C05469=1228.924,245.140,-60.585,-176.917,6.303,148.228
C05470=1228.928,244.891,-60.559,-176.919,6.301,148.228
C05471=1228.932,244.643,-60.532,-176.921,6.299,148.228
C05472=1228.937,244.394,-60.506,-176.924,6.297,148.229
C05473=1228.941,244.145,-60.480,-176.927,6.295,148.229
C05474=1228.945,243.897,-60.454,-176.929,6.293,148.229
C05475=1228.950,243.648,-60.428,-176.932,6.291,148.230
C05476=1228.955,243.399,-60.402,-176.934,6.289,148.230
C05477=1228.959,243.151,-60.376,-176.937,6.287,148.230
C05478=1228.963,242.902,-60.349,-176.939,6.285,148.230
C05479=1228.968,242.653,-60.323,-176.941,6.284,148.231
C05480=1228.972,242.405,-60.297,-176.944,6.282,148.231
C05481=1228.976,242.157,-60.272,-176.946,6.280,148.231
C05482=1228.981,241.908,-60.245,-176.949,6.278,148.231
C05483=1228.986,241.659,-60.220,-176.951,6.276,148.232
C05484=1228.990,241.411,-60.193,-176.954,6.275,148.232
C05485=1228.995,241.162,-60.167,-176.956,6.273,148.232
C05486=1228.999,240.914,-60.141,-176.959,6.271,148.233
C05487=1229.004,240.665,-60.116,-176.961,6.269,148.233
C05488=1229.008,240.416,-60.090,-176.964,6.267,148.233
C05489=1229.012,240.168,-60.063,-176.966,6.265,148.233
C05490=1229.017,239.920,-60.037,-176.969,6.263,148.234
C05491=1229.022,239.671,-60.012,-176.972,6.261,148.234
C05492=1229.026,239.422,-59.986,-176.974,6.259,148.234
C05493=1229.030,239.173,-59.960,-176.977,6.257,148.235
C05494=1229.036,238.925,-59.934,-176.979,6.255,148.235
C05495=1229.040,238.676,-59.908,-176.982,6.253,148.235
C05496=1229.044,238.428,-59.882,-176.984,6.251,148.235
C05497=1229.048,238.179,-59.856,-176.987,6.250,148.236
C05498=1229.053,237.908,-59.828,-176.990,6.248,148.236
C05499=1229.058,237.636,-59.800,-176.992,6.246,148.236
C05500=1229.063,237.365,-59.772,-176.995,6.244,148.237
C05501=1229.068,237.093,-59.744,-176.997,6.242,148.237
C05502=1229.073,236.844,-59.718,-177.000,6.240,148.237
C05503=1229.077,236.596,-59.692,-177.003,6.238,148.238
C05504=1229.082,236.347,-59.667,-177.005,6.236,148.238
C05505=1229.086,236.099,-59.641,-177.008,6.235,148.238
C05506=1229.090,235.850,-59.615,-177.010,6.232,148.238
C05507=1229.095,235.602,-59.590,-177.013,6.230,148.239
C05508=1229.099,235.353,-59.564,-177.015,6.229,148.239
C05509=1229.103,235.104,-59.538,-177.018,6.227,148.239
C05510=1229.108,234.856,-59.513,-177.020,6.225,148.240
C05511=1229.113,234.607,-59.486,-177.023,6.223,148.240
C05512=1229.117,234.358,-59.461,-177.026,6.221,148.240
C05513=1229.122,234.110,-59.435,-177.028,6.219,148.241
C05514=1229.126,233.861,-59.410,-177.031,6.217,148.241
C05515=1229.131,233.612,-59.384,-177.032,6.216,148.241
C05516=1229.136,233.364,-59.359,-177.035,6.214,148.241
C05517=1229.140,233.115,-59.333,-177.038,6.212,148.242
C05518=1229.144,232.866,-59.308,-177.040,6.210,148.242
C05519=1229.149,232.618,-59.282,-177.043,6.208,148.242
C05520=1229.153,232.369,-59.256,-177.046,6.207,148.243
C05521=1229.157,232.120,-59.231,-177.048,6.205,148.243
C05522=1229.163,231.872,-59.206,-177.051,6.203,148.243
C05523=1229.167,231.623,-59.180,-177.053,6.201,148.244
C05524=1229.172,231.375,-59.155,-177.056,6.199,148.244
C05525=1229.176,231.126,-59.129,-177.059,6.197,148.244
C05526=1229.180,230.877,-59.103,-177.060,6.196,148.244
C05527=1229.185,230.628,-59.079,-177.063,6.194,148.245
C05528=1229.189,230.379,-59.053,-177.066,6.192,148.245
C05529=1229.194,230.131,-59.028,-177.068,6.190,148.245
C05530=1229.199,229.882,-59.003,-177.071,6.188,148.246
C05531=1229.202,229.633,-58.977,-177.073,6.186,148.246
C05532=1229.207,229.385,-58.952,-177.076,6.185,148.246
C05533=1229.211,229.137,-58.926,-177.079,6.183,148.247
C05534=1229.216,228.888,-58.902,-177.081,6.181,148.247
C05535=1229.221,228.639,-58.876,-177.084,6.179,148.247
C05536=1229.225,228.390,-58.850,-177.086,6.178,148.248
C05537=1229.230,228.141,-58.825,-177.089,6.176,148.248
C05538=1229.234,227.893,-58.800,-177.091,6.174,148.248
C05539=1229.239,227.645,-58.774,-177.094,6.172,148.249
C05540=1229.244,227.395,-58.749,-177.096,6.170,148.249
C05541=1229.248,227.147,-58.724,-177.099,6.168,148.249
C05542=1229.252,226.898,-58.699,-177.101,6.166,148.249
C05543=1229.257,226.650,-58.674,-177.104,6.165,148.250
C05544=1229.261,226.401,-58.648,-177.106,6.163,148.250
C05545=1229.266,226.152,-58.624,-177.108,6.162,148.250
C05546=1229.271,225.903,-58.598,-177.111,6.160,148.251
C05547=1229.274,225.654,-58.573,-177.114,6.158,148.251
C05548=1229.279,225.406,-58.548,-177.116,6.156,148.251
C05549=1229.284,225.157,-58.523,-177.119,6.154,148.252
C05550=1229.289,224.909,-58.498,-177.122,6.152,148.252
C05551=1229.293,224.659,-58.473,-177.124,6.150,148.252
C05552=1229.297,224.412,-58.448,-177.127,6.149,148.253
C05553=1229.302,224.162,-58.423,-177.129,6.147,148.253
C05554=1229.307,223.914,-58.397,-177.132,6.146,148.253
C05555=1229.311,223.665,-58.372,-177.134,6.144,148.254
C05556=1229.315,223.417,-58.348,-177.137,6.142,148.254
C05557=1229.320,223.168,-58.323,-177.139,6.140,148.254
C05558=1229.325,222.919,-58.297,-177.142,6.138,148.255
C05559=1229.330,222.671,-58.272,-177.145,6.136,148.255
C05560=1229.333,222.421,-58.248,-177.147,6.134,148.255
C05561=1229.338,222.173,-58.223,-177.149,6.133,148.256
C05562=1229.343,221.924,-58.198,-177.152,6.132,148.256
C05563=1229.348,221.676,-58.172,-177.155,6.130,148.256
C05564=1229.351,221.427,-58.148,-177.157,6.128,148.257
C05565=1229.357,221.178,-58.123,-177.160,6.126,148.257
C05566=1229.361,220.929,-58.097,-177.162,6.124,148.257
C05567=1229.365,220.681,-58.073,-177.165,6.122,148.258
C05568=1229.370,220.432,-58.049,-177.168,6.120,148.258
C05569=1229.375,220.183,-58.023,-177.170,6.119,148.258
C05570=1229.379,219.935,-57.999,-177.172,6.117,148.259
C05571=1229.384,219.685,-57.974,-177.175,6.116,148.259
C05572=1229.388,219.437,-57.950,-177.178,6.114,148.259
C05573=1229.392,219.188,-57.924,-177.180,6.112,148.260
C05574=1229.397,218.939,-57.899,-177.183,6.110,148.260
C05575=1229.402,218.691,-57.875,-177.186,6.108,148.260
C05576=1229.406,218.442,-57.850,-177.188,6.107,148.261
C05577=1229.411,218.193,-57.825,-177.190,6.105,148.261
C05578=1229.415,217.944,-57.800,-177.193,6.103,148.261
C05579=1229.420,217.696,-57.776,-177.196,6.101,148.262
C05580=1229.424,217.447,-57.752,-177.198,6.100,148.262
C05581=1229.429,217.198,-57.727,-177.201,6.098,148.262
C05582=1229.433,216.950,-57.702,-177.203,6.096,148.263
C05583=1229.438,216.701,-57.677,-177.205,6.095,148.263
C05584=1229.443,216.452,-57.652,-177.208,6.093,148.263
C05585=1229.447,216.203,-57.628,-177.211,6.091,148.264
C05586=1229.452,215.955,-57.603,-177.213,6.089,148.264
C05587=1229.456,215.706,-57.579,-177.216,6.087,148.264
C05588=1229.461,215.457,-57.554,-177.219,6.086,148.265
C05589=1229.465,215.209,-57.529,-177.221,6.085,148.265
C05590=1229.470,214.960,-57.504,-177.223,6.083,148.265
C05591=1229.474,214.711,-57.480,-177.226,6.081,148.266
C05592=1229.479,214.463,-57.456,-177.229,6.079,148.266
C05593=1229.483,214.213,-57.431,-177.232,6.077,148.266
C05594=1229.488,213.965,-57.407,-177.234,6.076,148.267
C05595=1229.493,213.716,-57.382,-177.236,6.074,148.267
C05596=1229.497,213.467,-57.357,-177.239,6.073,148.267
C05597=1229.501,213.218,-57.333,-177.242,6.071,148.268
C05598=1229.507,212.970,-57.309,-177.244,6.069,148.268
C05599=1229.510,212.721,-57.284,-177.247,6.067,148.268
C05600=1229.515,212.472,-57.260,-177.250,6.065,148.269
C05601=1229.520,212.223,-57.235,-177.252,6.064,148.269
C05602=1229.525,211.953,-57.209,-177.254,6.062,148.270
C05603=1229.530,211.682,-57.182,-177.257,6.061,148.270
C05604=1229.534,211.412,-57.156,-177.261,6.058,148.270
C05605=1229.539,211.142,-57.130,-177.263,6.056,148.271
C05606=1229.545,210.893,-57.105,-177.265,6.055,148.271
C05607=1229.548,210.644,-57.080,-177.268,6.053,148.271
C05608=1229.553,210.396,-57.056,-177.270,6.051,148.272
C05609=1229.558,210.147,-57.032,-177.273,6.050,148.272
C05610=1229.563,209.898,-57.008,-177.276,6.048,148.272
C05611=1229.566,209.649,-56.984,-177.278,6.047,148.273
C05612=1229.572,209.400,-56.959,-177.281,6.045,148.273
C05613=1229.576,209.152,-56.935,-177.284,6.043,148.274
C05614=1229.580,208.903,-56.911,-177.286,6.041,148.274
C05615=1229.585,208.654,-56.886,-177.289,6.040,148.274
C05616=1229.590,208.405,-56.863,-177.291,6.039,148.275
C05617=1229.594,208.156,-56.839,-177.294,6.037,148.275
C05618=1229.599,207.908,-56.814,-177.296,6.035,148.275
C05619=1229.603,207.659,-56.790,-177.299,6.033,148.276
C05620=1229.608,207.411,-56.766,-177.301,6.031,148.276
C05621=1229.613,207.161,-56.742,-177.304,6.030,148.276
C05622=1229.617,206.912,-56.717,-177.306,6.028,148.277
C05623=1229.621,206.664,-56.693,-177.309,6.027,148.277
C05624=1229.626,206.415,-56.670,-177.312,6.025,148.278
C05625=1229.631,206.166,-56.645,-177.314,6.024,148.278
C05626=1229.635,205.917,-56.621,-177.317,6.022,148.278
C05627=1229.640,205.669,-56.597,-177.319,6.020,148.279
C05628=1229.644,205.420,-56.573,-177.322,6.018,148.279
C05629=1229.649,205.171,-56.549,-177.325,6.016,148.279
C05630=1229.654,204.922,-56.525,-177.327,6.015,148.280
C05631=1229.658,204.673,-56.501,-177.329,6.014,148.280
C05632=1229.662,204.424,-56.477,-177.332,6.012,148.280
C05633=1229.667,204.176,-56.452,-177.335,6.010,148.281
C05634=1229.672,203.926,-56.429,-177.337,6.009,148.281
C05635=1229.676,203.678,-56.405,-177.340,6.007,148.282
C05636=1229.681,203.429,-56.381,-177.342,6.005,148.282
C05637=1229.686,203.181,-56.357,-177.345,6.004,148.282
C05638=1229.690,202.932,-56.333,-177.347,6.003,148.283
C05639=1229.695,202.683,-56.309,-177.350,6.001,148.283
C05640=1229.699,202.434,-56.285,-177.352,5.999,148.283
C05641=1229.704,202.185,-56.262,-177.355,5.997,148.284
C05642=1229.708,201.936,-56.237,-177.358,5.996,148.284
C05643=1229.713,201.687,-56.214,-177.360,5.994,148.285
C05644=1229.717,201.439,-56.190,-177.363,5.993,148.285
C05645=1229.722,201.190,-56.167,-177.365,5.991,148.285
C05646=1229.727,200.941,-56.142,-177.368,5.990,148.286
C05647=1229.732,200.692,-56.119,-177.370,5.988,148.286
C05648=1229.736,200.444,-56.095,-177.373,5.986,148.286
C05649=1229.741,200.195,-56.071,-177.376,5.984,148.287
C05650=1229.745,199.946,-56.047,-177.378,5.983,148.287
C05651=1229.749,199.696,-56.023,-177.381,5.982,148.288
C05652=1229.754,199.448,-55.999,-177.383,5.980,148.288
C05653=1229.759,199.199,-55.976,-177.386,5.978,148.288
C05654=1229.763,198.950,-55.953,-177.388,5.977,148.289
C05655=1229.768,198.702,-55.929,-177.391,5.975,148.289
C05656=1229.772,198.453,-55.905,-177.394,5.973,148.290
C05657=1229.777,198.204,-55.881,-177.396,5.972,148.290
C05658=1229.781,197.955,-55.858,-177.398,5.971,148.290
C05659=1229.786,197.706,-55.834,-177.401,5.969,148.291
C05660=1229.791,197.458,-55.810,-177.404,5.967,148.291
C05661=1229.795,197.209,-55.787,-177.406,5.966,148.291
C05662=1229.800,196.960,-55.764,-177.408,5.964,148.292
C05663=1229.804,196.711,-55.740,-177.412,5.962,148.292
C05664=1229.809,196.462,-55.716,-177.414,5.961,148.293
C05665=1229.814,196.213,-55.693,-177.416,5.960,148.293
C05666=1229.818,195.964,-55.669,-177.419,5.958,148.293
C05667=1229.823,195.716,-55.645,-177.422,5.956,148.294
C05668=1229.828,195.467,-55.622,-177.424,5.955,148.294
C05669=1229.832,195.218,-55.599,-177.427,5.953,148.295
C05670=1229.837,194.969,-55.575,-177.429,5.951,148.295
C05671=1229.841,194.720,-55.551,-177.432,5.950,148.295
C05672=1229.846,194.471,-55.528,-177.434,5.949,148.296
C05673=1229.851,194.222,-55.505,-177.437,5.947,148.296
C05674=1229.855,193.973,-55.481,-177.439,5.945,148.296
C05675=1229.860,193.725,-55.457,-177.442,5.944,148.297
C05676=1229.865,193.476,-55.434,-177.445,5.942,148.297
C05677=1229.869,193.227,-55.410,-177.447,5.941,148.298
C05678=1229.873,192.978,-55.388,-177.449,5.940,148.298
C05679=1229.878,192.729,-55.364,-177.452,5.938,148.298
C05680=1229.883,192.480,-55.341,-177.455,5.936,148.299
C05681=1229.888,192.232,-55.317,-177.457,5.935,148.299
C05682=1229.892,191.983,-55.294,-177.460,5.933,148.300
C05683=1229.897,191.734,-55.270,-177.463,5.931,148.300
C05684=1229.902,191.485,-55.247,-177.465,5.930,148.300
C05685=1229.906,191.236,-55.224,-177.467,5.929,148.301
C05686=1229.910,190.987,-55.201,-177.470,5.927,148.301
C05687=1229.915,190.738,-55.178,-177.473,5.925,148.302
C05688=1229.920,190.489,-55.154,-177.475,5.924,148.302
C05689=1229.924,190.240,-55.131,-177.478,5.922,148.302
C05690=1229.929,189.991,-55.108,-177.480,5.920,148.303
C05691=1229.933,189.742,-55.085,-177.483,5.920,148.303
C05692=1229.938,189.494,-55.062,-177.486,5.918,148.304
C05693=1229.943,189.245,-55.038,-177.488,5.916,148.304
C05694=1229.948,188.996,-55.015,-177.490,5.915,148.304
C05695=1229.953,188.747,-54.992,-177.493,5.913,148.305
C05696=1229.956,188.498,-54.969,-177.496,5.912,148.305
C05697=1229.961,188.249,-54.946,-177.498,5.911,148.306
C05698=1229.966,188.000,-54.922,-177.501,5.909,148.306
C05699=1229.971,187.751,-54.899,-177.503,5.907,148.306
C05700=1229.975,187.503,-54.876,-177.506,5.906,148.307
C05701=1229.980,187.254,-54.853,-177.509,5.904,148.307
C05702=1229.985,187.005,-54.830,-177.511,5.903,148.308
C05703=1229.989,186.756,-54.806,-177.513,5.902,148.308
C05704=1229.993,186.507,-54.784,-177.516,5.900,148.309
C05705=1229.998,186.258,-54.760,-177.519,5.899,148.309
C05706=1230.003,185.989,-54.735,-177.521,5.897,148.309
C05707=1230.008,185.719,-54.711,-177.524,5.895,148.310
C05708=1230.013,185.449,-54.686,-177.527,5.894,148.310
C05709=1230.018,185.180,-54.661,-177.530,5.892,148.311
C05710=1230.022,184.931,-54.638,-177.532,5.890,148.311
C05711=1230.028,184.682,-54.615,-177.535,5.890,148.312
C05712=1230.033,184.433,-54.592,-177.538,5.888,148.312
C05713=1230.037,184.184,-54.570,-177.540,5.886,148.312
C05714=1230.041,183.935,-54.546,-177.542,5.885,148.313
C05715=1230.046,183.686,-54.523,-177.545,5.883,148.313
C05716=1230.051,183.438,-54.500,-177.548,5.882,148.314
C05717=1230.056,183.188,-54.478,-177.550,5.880,148.314
C05718=1230.060,182.940,-54.455,-177.553,5.879,148.314
C05719=1230.064,182.691,-54.432,-177.555,5.878,148.315
C05720=1230.069,182.442,-54.408,-177.558,5.876,148.315
C05721=1230.074,182.193,-54.387,-177.561,5.874,148.316
C05722=1230.079,181.944,-54.363,-177.563,5.873,148.316
C05723=1230.083,181.695,-54.341,-177.566,5.872,148.317
C05724=1230.088,181.446,-54.318,-177.568,5.871,148.317
C05725=1230.092,181.198,-54.295,-177.571,5.869,148.317
C05726=1230.097,180.948,-54.272,-177.573,5.867,148.318
C05727=1230.102,180.699,-54.249,-177.576,5.866,148.318
C05728=1230.106,180.450,-54.227,-177.579,5.864,148.319
C05729=1230.111,180.202,-54.204,-177.581,5.863,148.319
C05730=1230.115,179.952,-54.182,-177.583,5.862,148.319
C05731=1230.120,179.703,-54.158,-177.586,5.860,148.320
C05732=1230.125,179.455,-54.136,-177.589,5.859,148.320
C05733=1230.130,179.206,-54.113,-177.591,5.857,148.321
C05734=1230.134,178.957,-54.091,-177.593,5.856,148.321
C05735=1230.139,178.707,-54.068,-177.596,5.855,148.322
C05736=1230.143,178.459,-54.045,-177.599,5.853,148.322
C05737=1230.148,178.210,-54.022,-177.601,5.852,148.323
C05738=1230.152,177.961,-54.000,-177.604,5.850,148.323
C05739=1230.157,177.713,-53.977,-177.606,5.849,148.323
C05740=1230.162,177.463,-53.955,-177.609,5.848,148.324
C05741=1230.166,177.214,-53.932,-177.612,5.846,148.324
C05742=1230.171,176.966,-53.910,-177.614,5.845,148.325
C05743=1230.175,176.717,-53.887,-177.617,5.843,148.325
C05744=1230.180,176.467,-53.865,-177.619,5.842,148.326
C05745=1230.185,176.219,-53.842,-177.622,5.840,148.326
C05746=1230.190,175.970,-53.820,-177.625,5.839,148.326
C05747=1230.194,175.721,-53.797,-177.627,5.838,148.327
C05748=1230.199,175.472,-53.774,-177.629,5.836,148.327
C05749=1230.204,175.223,-53.752,-177.632,5.835,148.328
C05750=1230.208,174.974,-53.730,-177.635,5.833,148.328
C05751=1230.213,174.725,-53.707,-177.637,5.832,148.329
C05752=1230.217,174.476,-53.685,-177.639,5.831,148.329
C05753=1230.222,174.227,-53.662,-177.643,5.829,148.330
C05754=1230.227,173.979,-53.640,-177.645,5.828,148.330
C05755=1230.231,173.729,-53.618,-177.647,5.826,148.330
C05756=1230.237,173.480,-53.595,-177.650,5.826,148.331
C05757=1230.241,173.231,-53.573,-177.653,5.824,148.331
C05758=1230.245,172.982,-53.550,-177.655,5.823,148.332
C05759=1230.250,172.733,-53.528,-177.657,5.821,148.332
C05760=1230.254,172.484,-53.505,-177.660,5.819,148.333
C05761=1230.259,172.236,-53.484,-177.663,5.818,148.333
C05762=1230.264,171.986,-53.461,-177.665,5.817,148.333
C05763=1230.268,171.737,-53.438,-177.668,5.816,148.334
C05764=1230.273,171.489,-53.417,-177.670,5.814,148.334
C05765=1230.278,171.239,-53.394,-177.673,5.813,148.335
C05766=1230.283,170.991,-53.372,-177.676,5.812,148.335
C05767=1230.287,170.742,-53.350,-177.678,5.811,148.336
C05768=1230.292,170.493,-53.328,-177.680,5.809,148.336
C05769=1230.297,170.244,-53.305,-177.684,5.807,148.337
C05770=1230.301,169.994,-53.283,-177.686,5.806,148.337
C05771=1230.306,169.746,-53.261,-177.688,5.804,148.337
C05772=1230.310,169.497,-53.239,-177.691,5.804,148.338
C05773=1230.316,169.248,-53.216,-177.694,5.802,148.338
C05774=1230.320,168.999,-53.194,-177.696,5.801,148.339
C05775=1230.325,168.750,-53.173,-177.698,5.799,148.339
C05776=1230.329,168.501,-53.150,-177.701,5.798,148.340
C05777=1230.334,168.252,-53.128,-177.704,5.797,148.340
C05778=1230.338,168.003,-53.106,-177.706,5.796,148.340
C05779=1230.343,167.754,-53.084,-177.709,5.794,148.341
C05780=1230.348,167.505,-53.062,-177.711,5.793,148.341
C05781=1230.352,167.256,-53.040,-177.714,5.791,148.342
C05782=1230.358,167.007,-53.018,-177.717,5.790,148.342
C05783=1230.362,166.758,-52.996,-177.719,5.789,148.343
C05784=1230.366,166.509,-52.973,-177.721,5.787,148.343
C05785=1230.371,166.261,-52.951,-177.724,5.786,148.344
C05786=1230.375,166.011,-52.929,-177.727,5.784,148.344
C05787=1230.380,165.763,-52.908,-177.729,5.784,148.345
C05788=1230.385,165.513,-52.885,-177.732,5.782,148.345
C05789=1230.390,165.264,-52.863,-177.734,5.781,148.345
C05790=1230.394,165.015,-52.841,-177.737,5.779,148.346
C05791=1230.399,164.766,-52.820,-177.739,5.778,148.346
C05792=1230.404,164.517,-52.798,-177.742,5.777,148.347
C05793=1230.408,164.268,-52.776,-177.744,5.776,148.347
C05794=1230.413,164.019,-52.754,-177.747,5.774,148.348
C05795=1230.418,163.770,-52.732,-177.749,5.773,148.348
C05796=1230.422,163.521,-52.710,-177.752,5.772,148.349
C05797=1230.427,163.272,-52.688,-177.754,5.771,148.349
C05798=1230.432,163.023,-52.666,-177.757,5.769,148.349
C05799=1230.437,162.774,-52.644,-177.760,5.768,148.350
C05800=1230.442,162.525,-52.622,-177.762,5.766,148.350
C05801=1230.446,162.276,-52.600,-177.764,5.765,148.351
C05802=1230.451,162.027,-52.579,-177.768,5.764,148.351
C05803=1230.455,161.778,-52.557,-177.770,5.763,148.352
C05804=1230.460,161.529,-52.536,-177.773,5.761,148.352
C05805=1230.465,161.280,-52.514,-177.775,5.760,148.353
C05806=1230.469,161.031,-52.492,-177.778,5.758,148.353
C05807=1230.474,160.782,-52.470,-177.780,5.758,148.354
C05808=1230.478,160.533,-52.448,-177.783,5.756,148.354
C05809=1230.483,160.284,-52.427,-177.785,5.755,148.355
C05810=1230.489,160.015,-52.403,-177.788,5.753,148.355
C05811=1230.493,159.746,-52.380,-177.791,5.752,148.356
C05812=1230.499,159.477,-52.356,-177.793,5.751,148.356
C05813=1230.503,159.208,-52.334,-177.797,5.749,148.357
C05814=1230.508,158.959,-52.312,-177.799,5.748,148.357
C05815=1230.513,158.710,-52.290,-177.801,5.747,148.358
C05816=1230.517,158.461,-52.268,-177.804,5.746,148.358
C05817=1230.522,158.211,-52.247,-177.807,5.744,148.358
C05818=1230.527,157.963,-52.225,-177.809,5.743,148.359
C05819=1230.531,157.714,-52.203,-177.812,5.742,148.359
C05820=1230.536,157.465,-52.181,-177.814,5.741,148.360
C05821=1230.541,157.216,-52.160,-177.817,5.739,148.360
C05822=1230.545,156.966,-52.138,-177.819,5.738,148.361
C05823=1230.550,156.718,-52.117,-177.822,5.737,148.361
C05824=1230.555,156.468,-52.096,-177.824,5.736,148.362
C05825=1230.560,156.219,-52.074,-177.826,5.735,148.362
C05826=1230.565,155.970,-52.052,-177.830,5.733,148.363
C05827=1230.569,155.721,-52.032,-177.832,5.732,148.363
C05828=1230.574,155.473,-52.010,-177.835,5.731,148.364
C05829=1230.578,155.223,-51.988,-177.837,5.730,148.364
C05830=1230.583,154.974,-51.967,-177.840,5.728,148.365
C05831=1230.588,154.726,-51.945,-177.842,5.727,148.365
C05832=1230.592,154.476,-51.923,-177.845,5.725,148.366
C05833=1230.598,154.227,-51.902,-177.848,5.725,148.366
C05834=1230.602,153.979,-51.881,-177.850,5.723,148.367
C05835=1230.606,153.729,-51.860,-177.852,5.722,148.367
C05836=1230.611,153.480,-51.838,-177.855,5.721,148.368
C05837=1230.616,153.231,-51.817,-177.858,5.719,148.368
C05838=1230.621,152.982,-51.796,-177.860,5.719,148.369
C05839=1230.626,152.733,-51.773,-177.863,5.717,148.369
C05840=1230.630,152.484,-51.753,-177.865,5.716,148.370
C05841=1230.635,152.235,-51.731,-177.868,5.714,148.370
C05842=1230.640,151.986,-51.710,-177.870,5.713,148.370
C05843=1230.644,151.737,-51.688,-177.873,5.712,148.371
C05844=1230.649,151.488,-51.668,-177.875,5.711,148.371
C05845=1230.654,151.239,-51.646,-177.878,5.710,148.372
C05846=1230.659,150.990,-51.625,-177.881,5.709,148.372
C05847=1230.663,150.740,-51.603,-177.883,5.708,148.373
C05848=1230.667,150.491,-51.583,-177.886,5.706,148.373
C05849=1230.672,150.243,-51.561,-177.888,5.705,148.374
C05850=1230.678,149.994,-51.540,-177.891,5.704,148.374
C05851=1230.682,149.744,-51.518,-177.893,5.703,148.375
C05852=1230.686,149.495,-51.498,-177.896,5.702,148.375
C05853=1230.691,149.246,-51.477,-177.899,5.700,148.376
C05854=1230.696,148.997,-51.455,-177.901,5.699,148.376
C05855=1230.701,148.748,-51.434,-177.904,5.698,148.377
C05856=1230.705,148.499,-51.413,-177.906,5.697,148.377
C05857=1230.710,148.250,-51.392,-177.908,5.696,148.378
C05858=1230.715,148.001,-51.371,-177.911,5.694,148.378
C05859=1230.719,147.752,-51.350,-177.914,5.693,148.379
C05860=1230.725,147.503,-51.329,-177.916,5.692,148.379
C05861=1230.730,147.254,-51.308,-177.919,5.691,148.380
C05862=1230.733,147.005,-51.286,-177.921,5.690,148.380
C05863=1230.739,146.755,-51.265,-177.924,5.689,148.381
C05864=1230.744,146.506,-51.245,-177.926,5.688,148.381
C05865=1230.748,146.258,-51.223,-177.930,5.686,148.382
C05866=1230.753,146.009,-51.202,-177.932,5.685,148.382
C05867=1230.757,145.760,-51.182,-177.934,5.684,148.383
C05868=1230.762,145.510,-51.160,-177.937,5.683,148.383
C05869=1230.767,145.261,-51.139,-177.939,5.682,148.384
C05870=1230.771,145.012,-51.119,-177.942,5.680,148.384
C05871=1230.776,144.763,-51.098,-177.944,5.679,148.385
C05872=1230.781,144.514,-51.077,-177.947,5.678,148.385
C05873=1230.786,144.265,-51.056,-177.950,5.677,148.386
C05874=1230.790,144.016,-51.035,-177.952,5.676,148.386
C05875=1230.795,143.766,-51.014,-177.955,5.674,148.387
C05876=1230.800,143.517,-50.993,-177.957,5.674,148.387
C05877=1230.804,143.269,-50.972,-177.959,5.673,148.388
C05878=1230.809,143.019,-50.951,-177.963,5.671,148.388
C05879=1230.814,142.771,-50.931,-177.965,5.670,148.389
C05880=1230.819,142.521,-50.910,-177.967,5.669,148.389
C05881=1230.823,142.272,-50.889,-177.970,5.668,148.390
C05882=1230.829,142.023,-50.868,-177.973,5.667,148.390
C05883=1230.833,141.775,-50.847,-177.975,5.665,148.391
C05884=1230.838,141.525,-50.826,-177.978,5.665,148.391
C05885=1230.842,141.276,-50.805,-177.980,5.664,148.392
C05886=1230.847,141.027,-50.785,-177.983,5.662,148.392
C05887=1230.851,140.778,-50.764,-177.985,5.661,148.393
C05888=1230.856,140.528,-50.743,-177.987,5.660,148.393
C05889=1230.861,140.279,-50.723,-177.991,5.659,148.394
C05890=1230.866,140.030,-50.702,-177.993,5.658,148.394
C05891=1230.870,139.781,-50.681,-177.996,5.656,148.395
C05892=1230.876,139.532,-50.660,-177.998,5.655,148.395
C05893=1230.880,139.283,-50.640,-178.000,5.655,148.396
C05894=1230.885,139.034,-50.619,-178.003,5.653,148.396
C05895=1230.890,138.785,-50.599,-178.006,5.652,148.397
C05896=1230.894,138.536,-50.578,-178.008,5.651,148.397
C05897=1230.899,138.287,-50.557,-178.011,5.650,148.398
C05898=1230.904,138.038,-50.537,-178.013,5.649,148.398
C05899=1230.909,137.788,-50.516,-178.016,5.648,148.399
C05900=1230.913,137.539,-50.496,-178.018,5.646,148.399
C05901=1230.919,137.290,-50.475,-178.021,5.646,148.400
C05902=1230.923,137.041,-50.454,-178.023,5.645,148.400
C05903=1230.927,136.792,-50.434,-178.026,5.643,148.401
C05904=1230.933,136.543,-50.413,-178.028,5.642,148.401
C05905=1230.937,136.294,-50.393,-178.031,5.641,148.402
C05906=1230.941,136.045,-50.372,-178.034,5.640,148.402
C05907=1230.947,135.796,-50.351,-178.036,5.639,148.403
C05908=1230.951,135.547,-50.331,-178.039,5.638,148.403
C05909=1230.956,135.298,-50.311,-178.042,5.637,148.404
C05910=1230.961,135.049,-50.290,-178.044,5.636,148.404
C05911=1230.965,134.799,-50.270,-178.046,5.635,148.405
C05912=1230.971,134.550,-50.249,-178.049,5.633,148.405
C05913=1230.975,134.301,-50.229,-178.052,5.632,148.406
C05914=1230.980,134.033,-50.206,-178.055,5.631,148.406
C05915=1230.985,133.763,-50.185,-178.057,5.630,148.407
C05916=1230.990,133.495,-50.162,-178.060,5.628,148.407
C05917=1230.996,133.226,-50.141,-178.063,5.628,148.408
C05918=1231.000,132.977,-50.120,-178.065,5.627,148.409
C05919=1231.005,132.728,-50.100,-178.068,5.625,148.409
C05920=1231.010,132.479,-50.079,-178.070,5.625,148.410
C05921=1231.014,132.230,-50.059,-178.073,5.624,148.410
C05922=1231.019,131.980,-50.039,-178.076,5.622,148.411
C05923=1231.023,131.731,-50.019,-178.078,5.621,148.411
C05924=1231.029,131.482,-49.998,-178.080,5.621,148.412
C05925=1231.033,131.233,-49.977,-178.083,5.619,148.412
C05926=1231.038,130.984,-49.958,-178.086,5.618,148.413
C05927=1231.043,130.735,-49.938,-178.088,5.617,148.413
C05928=1231.048,130.486,-49.917,-178.091,5.616,148.414
C05929=1231.053,130.236,-49.897,-178.094,5.615,148.414
C05930=1231.057,129.987,-49.877,-178.096,5.614,148.415
C05931=1231.062,129.739,-49.856,-178.099,5.613,148.415
C05932=1231.066,129.490,-49.836,-178.101,5.612,148.416
C05933=1231.071,129.240,-49.816,-178.104,5.611,148.417
C05934=1231.076,128.991,-49.795,-178.106,5.610,148.417
C05935=1231.081,128.742,-49.776,-178.109,5.609,148.418
C05936=1231.086,128.493,-49.756,-178.111,5.608,148.418
C05937=1231.090,128.244,-49.735,-178.114,5.607,148.419
C05938=1231.095,127.994,-49.716,-178.116,5.605,148.419
C05939=1231.100,127.745,-49.695,-178.119,5.605,148.420
C05940=1231.104,127.496,-49.674,-178.121,5.604,148.420
C05941=1231.109,127.247,-49.655,-178.124,5.603,148.421
C05942=1231.114,126.998,-49.634,-178.127,5.601,148.421
C05943=1231.119,126.749,-49.615,-178.129,5.601,148.422
C05944=1231.123,126.500,-49.595,-178.131,5.600,148.422
C05945=1231.128,126.250,-49.575,-178.134,5.598,148.423
C05946=1231.133,126.001,-49.554,-178.137,5.597,148.423
C05947=1231.138,125.751,-49.534,-178.139,5.597,148.424
C05948=1231.143,125.503,-49.514,-178.141,5.596,148.424
C05949=1231.148,125.254,-49.495,-178.145,5.594,148.425
C05950=1231.152,125.005,-49.474,-178.147,5.593,148.425
C05951=1231.157,124.755,-49.455,-178.149,5.593,148.426
C05952=1231.162,124.506,-49.434,-178.152,5.591,148.426
C05953=1231.166,124.257,-49.415,-178.155,5.590,148.427
C05954=1231.171,124.008,-49.395,-178.157,5.590,148.428
C05955=1231.176,123.759,-49.375,-178.159,5.589,148.428
C05956=1231.180,123.510,-49.354,-178.163,5.587,148.429
C05957=1231.185,123.260,-49.335,-178.165,5.586,148.429
C05958=1231.190,123.011,-49.314,-178.167,5.586,148.430
C05959=1231.195,122.762,-49.295,-178.170,5.585,148.430
C05960=1231.199,122.514,-49.275,-178.173,5.583,148.431
C05961=1231.204,122.264,-49.255,-178.175,5.583,148.431
C05962=1231.209,122.014,-49.235,-178.177,5.582,148.432
C05963=1231.214,121.766,-49.215,-178.180,5.581,148.432
C05964=1231.219,121.517,-49.196,-178.183,5.579,148.433
C05965=1231.223,121.267,-49.176,-178.185,5.579,148.434
C05966=1231.228,121.018,-49.156,-178.188,5.578,148.434
C05967=1231.233,120.769,-49.136,-178.190,5.577,148.435
C05968=1231.238,120.520,-49.117,-178.193,5.575,148.435
C05969=1231.242,120.271,-49.096,-178.195,5.574,148.436
C05970=1231.247,120.021,-49.077,-178.198,5.574,148.436
C05971=1231.252,119.772,-49.058,-178.200,5.573,148.437
C05972=1231.257,119.523,-49.037,-178.203,5.571,148.437
C05973=1231.262,119.274,-49.017,-178.206,5.571,148.438
C05974=1231.266,119.024,-48.998,-178.208,5.570,148.438
C05975=1231.271,118.776,-48.978,-178.210,5.569,148.439
C05976=1231.276,118.526,-48.958,-178.214,5.568,148.440
C05977=1231.281,118.277,-48.939,-178.216,5.567,148.440
C05978=1231.286,118.028,-48.919,-178.218,5.566,148.441
C05979=1231.291,117.779,-48.899,-178.220,5.565,148.441
C05980=1231.295,117.530,-48.880,-178.224,5.564,148.442
C05981=1231.300,117.281,-48.861,-178.226,5.563,148.442
C05982=1231.305,117.031,-48.841,-178.228,5.562,148.443
C05983=1231.310,116.782,-48.821,-178.231,5.561,148.443
C05984=1231.314,116.533,-48.801,-178.234,5.560,148.444
C05985=1231.319,116.284,-48.782,-178.236,5.559,148.444
C05986=1231.324,116.034,-48.762,-178.239,5.558,148.445
C05987=1231.329,115.785,-48.742,-178.241,5.557,148.445
C05988=1231.333,115.536,-48.724,-178.244,5.557,148.446
C05989=1231.338,115.287,-48.704,-178.247,5.555,148.447
C05990=1231.343,115.038,-48.684,-178.249,5.554,148.447
C05991=1231.348,114.789,-48.664,-178.251,5.554,148.448
C05992=1231.353,114.539,-48.645,-178.254,5.553,148.448
C05993=1231.358,114.290,-48.625,-178.257,5.551,148.449
C05994=1231.362,114.041,-48.606,-178.259,5.551,148.449
C05995=1231.367,113.792,-48.587,-178.261,5.550,148.450
C05996=1231.372,113.543,-48.567,-178.264,5.549,148.450
C05997=1231.377,113.293,-48.548,-178.267,5.548,148.451
C05998=1231.382,113.044,-48.528,-178.269,5.547,148.452
C05999=1231.386,112.795,-48.509,-178.272,5.546,148.452
C06000=1231.391,112.545,-48.490,-178.275,5.545,148.453
C06001=1231.396,112.297,-48.470,-178.277,5.544,148.453
C06002=1231.401,112.048,-48.450,-178.279,5.544,148.454
C06003=1231.405,111.798,-48.431,-178.283,5.542,148.454
C06004=1231.410,111.549,-48.412,-178.285,5.541,148.455
C06005=1231.415,111.300,-48.392,-178.287,5.541,148.456
C06006=1231.420,111.051,-48.373,-178.290,5.540,148.456
C06007=1231.424,110.802,-48.354,-178.292,5.539,148.457
C06008=1231.429,110.552,-48.335,-178.295,5.538,148.457
C06009=1231.435,110.303,-48.315,-178.297,5.537,148.458
C06010=1231.439,110.053,-48.296,-178.300,5.536,148.458
C06011=1231.444,109.805,-48.277,-178.302,5.536,148.459
C06012=1231.449,109.555,-48.257,-178.305,5.535,148.459
C06013=1231.454,109.306,-48.238,-178.308,5.533,148.460
C06014=1231.458,109.057,-48.219,-178.310,5.532,148.461
C06015=1231.463,108.807,-48.199,-178.313,5.532,148.461
C06016=1231.468,108.558,-48.180,-178.315,5.531,148.462
C06017=1231.472,108.309,-48.161,-178.318,5.530,148.462
C06018=1231.478,108.041,-48.140,-178.321,5.529,148.463
C06019=1231.483,107.772,-48.120,-178.323,5.528,148.463
C06020=1231.488,107.504,-48.099,-178.326,5.527,148.464
C06021=1231.493,107.235,-48.078,-178.329,5.526,148.465
C06022=1231.498,106.987,-48.059,-178.331,5.525,148.465
C06023=1231.503,106.737,-48.040,-178.334,5.525,148.466
C06024=1231.508,106.488,-48.021,-178.336,5.524,148.466
C06025=1231.512,106.239,-48.002,-178.339,5.523,148.467
C06026=1231.518,105.990,-47.983,-178.342,5.522,148.468
C06027=1231.522,105.740,-47.963,-178.344,5.521,148.468
C06028=1231.526,105.491,-47.944,-178.347,5.520,148.469
C06029=1231.532,105.241,-47.925,-178.349,5.519,148.469
C06030=1231.536,104.992,-47.906,-178.351,5.518,148.470
C06031=1231.541,104.743,-47.887,-178.354,5.518,148.470
C06032=1231.546,104.495,-47.868,-178.357,5.516,148.471
C06033=1231.551,104.244,-47.850,-178.359,5.515,148.471
C06034=1231.556,103.996,-47.830,-178.362,5.515,148.472
C06035=1231.560,103.746,-47.811,-178.365,5.514,148.473
C06036=1231.566,103.497,-47.792,-178.367,5.513,148.473
C06037=1231.570,103.248,-47.774,-178.369,5.512,148.474
C06038=1231.575,102.999,-47.754,-178.373,5.511,148.474
C06039=1231.579,102.749,-47.735,-178.375,5.510,148.475
C06040=1231.585,102.500,-47.717,-178.377,5.509,148.475
C06041=1231.589,102.251,-47.698,-178.380,5.509,148.476
C06042=1231.594,102.002,-47.678,-178.382,5.508,148.477
C06043=1231.599,101.752,-47.660,-178.385,5.507,148.477
C06044=1231.604,101.503,-47.641,-178.387,5.507,148.478
C06045=1231.609,101.255,-47.622,-178.390,5.505,148.478
C06046=1231.614,101.004,-47.603,-178.393,5.504,148.479
C06047=1231.618,100.756,-47.584,-178.395,5.504,148.480
C06048=1231.623,100.506,-47.565,-178.398,5.503,148.480
C06049=1231.628,100.257,-47.547,-178.400,5.502,148.481
C06050=1231.633,100.008,-47.527,-178.403,5.501,148.481
C06051=1231.638,99.758,-47.509,-178.405,5.501,148.482
C06052=1231.643,99.509,-47.490,-178.408,5.499,148.482
C06053=1231.647,99.260,-47.471,-178.410,5.498,148.483
C06054=1231.652,99.011,-47.453,-178.413,5.498,148.484
C06055=1231.657,98.761,-47.433,-178.416,5.497,148.484
C06056=1231.662,98.512,-47.415,-178.418,5.496,148.485
C06057=1231.667,98.263,-47.396,-178.420,5.496,148.485
C06058=1231.671,98.014,-47.377,-178.423,5.495,148.486
C06059=1231.677,97.765,-47.358,-178.425,5.494,148.486
C06060=1231.681,97.515,-47.340,-178.428,5.493,148.487
C06061=1231.685,97.266,-47.321,-178.431,5.492,148.488
C06062=1231.691,97.017,-47.302,-178.433,5.491,148.488
C06063=1231.695,96.768,-47.283,-178.436,5.490,148.489
C06064=1231.700,96.518,-47.265,-178.438,5.490,148.489
C06065=1231.705,96.269,-47.246,-178.441,5.489,148.490
C06066=1231.710,96.020,-47.228,-178.443,5.488,148.490
C06067=1231.715,95.770,-47.209,-178.446,5.488,148.491
C06068=1231.720,95.522,-47.191,-178.449,5.486,148.492
C06069=1231.724,95.272,-47.172,-178.451,5.486,148.492
C06070=1231.730,95.023,-47.153,-178.454,5.485,148.493
C06071=1231.734,94.774,-47.135,-178.456,5.484,148.493
C06072=1231.738,94.524,-47.116,-178.459,5.483,148.494
C06073=1231.744,94.275,-47.097,-178.461,5.482,148.495
C06074=1231.749,94.026,-47.079,-178.464,5.482,148.495
C06075=1231.753,93.776,-47.060,-178.466,5.481,148.496
C06076=1231.758,93.527,-47.042,-178.469,5.481,148.496
C06077=1231.764,93.278,-47.024,-178.472,5.479,148.497
C06078=1231.768,93.029,-47.005,-178.474,5.478,148.498
C06079=1231.773,92.779,-46.987,-178.477,5.478,148.498
C06080=1231.778,92.530,-46.968,-178.479,5.477,148.499
C06081=1231.782,92.281,-46.949,-178.482,5.476,148.499
C06082=1231.787,92.031,-46.931,-178.484,5.475,148.500
C06083=1231.792,91.782,-46.913,-178.487,5.475,148.501
C06084=1231.797,91.533,-46.893,-178.489,5.474,148.501
C06085=1231.802,91.284,-46.875,-178.492,5.473,148.502
C06086=1231.807,91.034,-46.857,-178.494,5.473,148.502
C06087=1231.811,90.785,-46.839,-178.497,5.471,148.503
C06088=1231.816,90.536,-46.820,-178.499,5.470,148.503
C06089=1231.821,90.286,-46.802,-178.502,5.470,148.504
C06090=1231.826,90.037,-46.784,-178.505,5.469,148.505
C06091=1231.831,89.788,-46.766,-178.507,5.468,148.505
C06092=1231.835,89.539,-46.747,-178.509,5.467,148.506
C06093=1231.841,89.289,-46.728,-178.512,5.467,148.506
C06094=1231.846,89.040,-46.710,-178.515,5.466,148.507
C06095=1231.850,88.791,-46.692,-178.517,5.466,148.508
C06096=1231.855,88.541,-46.674,-178.519,5.465,148.508
C06097=1231.859,88.293,-46.655,-178.522,5.464,148.509
C06098=1231.865,88.043,-46.637,-178.525,5.463,148.509
C06099=1231.870,87.794,-46.619,-178.528,5.462,148.510
C06100=1231.874,87.544,-46.600,-178.530,5.461,148.511
C06101=1231.879,87.295,-46.582,-178.533,5.460,148.511
C06102=1231.884,87.046,-46.564,-178.535,5.460,148.512
C06103=1231.889,86.797,-46.546,-178.538,5.459,148.512
C06104=1231.894,86.548,-46.528,-178.540,5.459,148.513
C06105=1231.899,86.298,-46.509,-178.543,5.458,148.514
C06106=1231.904,86.049,-46.491,-178.545,5.457,148.514
C06107=1231.908,85.799,-46.473,-178.548,5.457,148.515
C06108=1231.913,85.550,-46.455,-178.550,5.456,148.515
C06109=1231.918,85.301,-46.437,-178.553,5.455,148.516
C06110=1231.923,85.051,-46.418,-178.555,5.454,148.517
C06111=1231.927,84.802,-46.401,-178.558,5.454,148.517
C06112=1231.932,84.553,-46.383,-178.560,5.453,148.518
C06113=1231.937,84.304,-46.365,-178.563,5.452,148.518
C06114=1231.942,84.054,-46.347,-178.566,5.451,148.519
C06115=1231.947,83.805,-46.329,-178.568,5.450,148.520
C06116=1231.952,83.555,-46.310,-178.571,5.450,148.520
C06117=1231.957,83.306,-46.292,-178.574,5.449,148.521
C06118=1231.962,83.057,-46.274,-178.576,5.448,148.521
C06119=1231.967,82.808,-46.256,-178.578,5.447,148.522
C06120=1231.972,82.558,-46.238,-178.581,5.447,148.523
C06121=1231.977,82.309,-46.220,-178.584,5.446,148.523
C06122=1231.982,82.041,-46.200,-178.586,5.446,148.524
C06123=1231.987,81.773,-46.181,-178.589,5.445,148.525
C06124=1231.992,81.504,-46.162,-178.592,5.444,148.525
C06125=1231.997,81.236,-46.142,-178.595,5.443,148.526
C06126=1232.002,80.987,-46.124,-178.597,5.442,148.526
C06127=1232.006,80.737,-46.106,-178.599,5.441,148.527
C06128=1232.011,80.488,-46.088,-178.602,5.441,148.528
C06129=1232.016,80.238,-46.071,-178.605,5.440,148.528
C06130=1232.021,79.989,-46.053,-178.607,5.440,148.529
C06131=1232.026,79.740,-46.035,-178.610,5.439,148.529
C06132=1232.031,79.491,-46.017,-178.612,5.438,148.530
C06133=1232.036,79.241,-45.999,-178.615,5.437,148.531
C06134=1232.041,78.992,-45.981,-178.617,5.437,148.531
C06135=1232.046,78.743,-45.963,-178.620,5.436,148.532
C06136=1232.051,78.494,-45.945,-178.622,5.435,148.532
C06137=1232.055,78.243,-45.927,-178.625,5.435,148.533
C06138=1232.060,77.994,-45.909,-178.627,5.434,148.534
C06139=1232.065,77.745,-45.891,-178.630,5.434,148.534
C06140=1232.070,77.496,-45.873,-178.633,5.433,148.535
C06141=1232.075,77.247,-45.855,-178.635,5.432,148.536
C06142=1232.080,76.997,-45.838,-178.637,5.431,148.536
C06143=1232.084,76.748,-45.820,-178.640,5.431,148.537
C06144=1232.089,76.499,-45.803,-178.643,5.430,148.538
C06145=1232.094,76.250,-45.785,-178.645,5.430,148.538
C06146=1232.100,76.000,-45.767,-178.647,5.429,148.539
C06147=1232.104,75.751,-45.749,-178.650,5.428,148.539
C06148=1232.109,75.502,-45.731,-178.653,5.427,148.540
C06149=1232.114,75.252,-45.713,-178.655,5.427,148.541
C06150=1232.119,75.003,-45.697,-178.658,5.426,148.541
C06151=1232.124,74.754,-45.679,-178.660,5.425,148.542
C06152=1232.129,74.505,-45.661,-178.663,5.425,148.542
C06153=1232.133,74.255,-45.643,-178.665,5.424,148.543
C06154=1232.139,74.006,-45.625,-178.668,5.424,148.544
C06155=1232.144,73.756,-45.607,-178.671,5.423,148.544
C06156=1232.148,73.508,-45.590,-178.673,5.422,148.545
C06157=1232.153,73.258,-45.573,-178.675,5.421,148.545
C06158=1232.158,73.009,-45.555,-178.678,5.421,148.546
C06159=1232.163,72.759,-45.537,-178.681,5.420,148.547
C06160=1232.168,72.510,-45.520,-178.683,5.420,148.547
C06161=1232.172,72.261,-45.502,-178.686,5.419,148.548
C06162=1232.177,72.011,-45.485,-178.688,5.418,148.549
C06163=1232.182,71.762,-45.467,-178.691,5.418,148.549
C06164=1232.187,71.513,-45.449,-178.693,5.417,148.550
C06165=1232.192,71.263,-45.432,-178.696,5.416,148.550
C06166=1232.197,71.014,-45.414,-178.698,5.416,148.551
C06167=1232.202,70.764,-45.397,-178.701,5.415,148.552
C06168=1232.207,70.515,-45.379,-178.703,5.414,148.552
C06169=1232.212,70.265,-45.362,-178.706,5.414,148.553
C06170=1232.216,70.016,-45.344,-178.709,5.413,148.554
C06171=1232.221,69.767,-45.326,-178.711,5.412,148.554
C06172=1232.226,69.517,-45.309,-178.714,5.412,148.555
C06173=1232.230,69.268,-45.292,-178.716,5.411,148.555
C06174=1232.236,69.019,-45.275,-178.719,5.410,148.556
C06175=1232.241,68.770,-45.257,-178.721,5.410,148.557
C06176=1232.246,68.520,-45.239,-178.724,5.409,148.557
C06177=1232.250,68.271,-45.222,-178.726,5.409,148.558
C06178=1232.255,68.021,-45.205,-178.729,5.408,148.559
C06179=1232.261,67.773,-45.187,-178.732,5.407,148.559
C06180=1232.265,67.523,-45.170,-178.734,5.407,148.560
C06181=1232.270,67.274,-45.152,-178.736,5.406,148.560
C06182=1232.275,67.024,-45.135,-178.739,5.405,148.561
C06183=1232.280,66.775,-45.118,-178.742,5.405,148.562
C06184=1232.285,66.525,-45.100,-178.744,5.404,148.562
C06185=1232.290,66.276,-45.083,-178.747,5.404,148.563
C06186=1232.294,66.027,-45.066,-178.750,5.403,148.564
C06187=1232.299,65.777,-45.049,-178.752,5.402,148.564
C06188=1232.304,65.528,-45.031,-178.754,5.401,148.565
C06189=1232.309,65.279,-45.014,-178.757,5.401,148.565
C06190=1232.315,65.029,-44.997,-178.760,5.400,148.566
C06191=1232.319,64.780,-44.980,-178.762,5.400,148.567
C06192=1232.324,64.531,-44.962,-178.765,5.399,148.567
C06193=1232.329,64.281,-44.945,-178.768,5.398,148.568
C06194=1232.333,64.032,-44.928,-178.770,5.398,148.568
C06195=1232.339,63.782,-44.910,-178.772,5.397,148.569
C06196=1232.343,63.533,-44.894,-178.775,5.396,148.570
C06197=1232.349,63.284,-44.876,-178.778,5.396,148.570
C06198=1232.353,63.035,-44.860,-178.780,5.395,148.571
C06199=1232.358,62.785,-44.842,-178.783,5.395,148.572
C06200=1232.363,62.536,-44.824,-178.785,5.395,148.572
C06201=1232.368,62.286,-44.808,-178.787,5.394,148.573
C06202=1232.373,62.036,-44.790,-178.790,5.393,148.574
C06203=1232.378,61.788,-44.774,-178.792,5.393,148.574
C06204=1232.383,61.538,-44.756,-178.795,5.392,148.575
C06205=1232.387,61.289,-44.739,-178.798,5.392,148.576
C06206=1232.393,61.039,-44.722,-178.800,5.391,148.576
C06207=1232.397,60.790,-44.705,-178.803,5.390,148.577
C06208=1232.402,60.541,-44.687,-178.805,5.389,148.577
C06209=1232.407,60.292,-44.671,-178.808,5.389,148.578
C06210=1232.412,60.042,-44.654,-178.810,5.388,148.579
C06211=1232.417,59.792,-44.637,-178.813,5.388,148.579
C06212=1232.422,59.543,-44.619,-178.816,5.387,148.580
C06213=1232.426,59.294,-44.603,-178.818,5.387,148.581
C06214=1232.432,59.045,-44.586,-178.821,5.386,148.581
C06215=1232.436,58.795,-44.569,-178.823,5.385,148.582
C06216=1232.442,58.545,-44.552,-178.826,5.384,148.582
C06217=1232.446,58.296,-44.535,-178.828,5.385,148.583
C06218=1232.452,58.048,-44.517,-178.830,5.384,148.584
C06219=1232.456,57.798,-44.501,-178.833,5.384,148.584
C06220=1232.461,57.548,-44.484,-178.836,5.383,148.585
C06221=1232.466,57.299,-44.467,-178.838,5.382,148.586
C06222=1232.471,57.050,-44.451,-178.841,5.382,148.586
C06223=1232.476,56.800,-44.433,-178.843,5.381,148.587
C06224=1232.481,56.551,-44.417,-178.846,5.381,148.588
C06225=1232.486,56.301,-44.399,-178.848,5.380,148.588
C06226=1232.491,56.033,-44.382,-178.851,5.379,148.589
C06227=1232.496,55.764,-44.363,-178.854,5.379,148.590
C06228=1232.502,55.496,-44.345,-178.857,5.378,148.590
C06229=1232.507,55.227,-44.327,-178.859,5.378,148.591
C06230=1232.512,54.978,-44.310,-178.862,5.377,148.592
C06231=1232.517,54.729,-44.294,-178.864,5.377,148.592
C06232=1232.522,54.479,-44.276,-178.867,5.376,148.593
C06233=1232.526,54.230,-44.260,-178.869,5.375,148.594
C06234=1232.531,53.981,-44.243,-178.872,5.374,148.594
C06235=1232.537,53.731,-44.226,-178.875,5.374,148.595
C06236=1232.541,53.482,-44.209,-178.877,5.373,148.596
C06237=1232.546,53.232,-44.193,-178.880,5.373,148.596
C06238=1232.551,52.983,-44.176,-178.882,5.373,148.597
C06239=1232.556,52.734,-44.159,-178.885,5.372,148.598
C06240=1232.560,52.484,-44.142,-178.887,5.372,148.598
C06241=1232.566,52.235,-44.126,-178.890,5.371,148.599
C06242=1232.571,51.986,-44.109,-178.892,5.370,148.599
C06243=1232.575,51.736,-44.092,-178.895,5.370,148.600
C06244=1232.581,51.487,-44.075,-178.897,5.369,148.601
C06245=1232.585,51.238,-44.059,-178.900,5.369,148.601
C06246=1232.590,50.988,-44.042,-178.902,5.368,148.602
C06247=1232.596,50.739,-44.025,-178.905,5.367,148.603
C06248=1232.601,50.489,-44.009,-178.907,5.368,148.603
C06249=1232.605,50.239,-43.992,-178.910,5.367,148.604
C06250=1232.610,49.991,-43.976,-178.912,5.367,148.605
C06251=1232.615,49.741,-43.959,-178.915,5.366,148.605
C06252=1232.620,49.491,-43.942,-178.917,5.365,148.606
C06253=1232.625,49.243,-43.926,-178.920,5.364,148.607
C06254=1232.629,48.993,-43.909,-178.923,5.364,148.607
C06255=1232.635,48.743,-43.893,-178.925,5.363,148.608
C06256=1232.640,48.494,-43.876,-178.928,5.363,148.609
C06257=1232.644,48.244,-43.860,-178.930,5.362,148.609
C06258=1232.650,47.996,-43.843,-178.932,5.362,148.610
C06259=1232.654,47.746,-43.827,-178.935,5.362,148.611
C06260=1232.659,47.496,-43.809,-178.938,5.361,148.611
C06261=1232.665,47.247,-43.794,-178.940,5.361,148.612
C06262=1232.669,46.997,-43.777,-178.943,5.360,148.613
C06263=1232.674,46.748,-43.761,-178.946,5.360,148.613
C06264=1232.679,46.499,-43.744,-178.948,5.359,148.614
C06265=1232.684,46.249,-43.728,-178.950,5.358,148.614
C06266=1232.689,46.000,-43.711,-178.953,5.358,148.615
C06267=1232.694,45.751,-43.695,-178.955,5.358,148.616
C06268=1232.699,45.502,-43.678,-178.958,5.357,148.616
C06269=1232.704,45.252,-43.662,-178.960,5.357,148.617
C06270=1232.708,45.002,-43.646,-178.963,5.356,148.618
C06271=1232.714,44.753,-43.629,-178.966,5.355,148.618
C06272=1232.719,44.503,-43.613,-178.968,5.355,148.619
C06273=1232.724,44.254,-43.597,-178.971,5.354,148.620
C06274=1232.728,44.005,-43.580,-178.973,5.355,148.620
C06275=1232.734,43.755,-43.564,-178.976,5.354,148.621
C06276=1232.738,43.506,-43.548,-178.978,5.353,148.622
C06277=1232.743,43.256,-43.531,-178.980,5.353,148.622
C06278=1232.748,43.007,-43.515,-178.983,5.352,148.623
C06279=1232.753,42.757,-43.498,-178.986,5.351,148.624
C06280=1232.758,42.508,-43.482,-178.988,5.351,148.624
C06281=1232.763,42.258,-43.466,-178.991,5.350,148.625
C06282=1232.768,42.009,-43.450,-178.993,5.351,148.626
C06283=1232.773,41.760,-43.433,-178.996,5.350,148.626
C06284=1232.778,41.511,-43.417,-178.998,5.349,148.627
C06285=1232.782,41.261,-43.401,-179.001,5.349,148.628
C06286=1232.788,41.012,-43.385,-179.004,5.348,148.628
C06287=1232.792,40.762,-43.368,-179.006,5.348,148.629
C06288=1232.798,40.513,-43.353,-179.009,5.347,148.630
C06289=1232.802,40.263,-43.336,-179.011,5.347,148.630
C06290=1232.807,40.015,-43.320,-179.014,5.347,148.631
C06291=1232.812,39.764,-43.304,-179.016,5.346,148.632
C06292=1232.817,39.516,-43.288,-179.018,5.345,148.632
C06293=1232.822,39.266,-43.272,-179.021,5.345,148.633
C06294=1232.827,39.017,-43.255,-179.024,5.344,148.633
C06295=1232.832,38.767,-43.239,-179.026,5.344,148.634
C06296=1232.837,38.518,-43.223,-179.028,5.344,148.635
C06297=1232.842,38.267,-43.207,-179.031,5.343,148.635
C06298=1232.847,38.019,-43.191,-179.034,5.343,148.636
C06299=1232.852,37.769,-43.175,-179.036,5.342,148.637
C06300=1232.857,37.520,-43.159,-179.039,5.342,148.637
C06301=1232.861,37.270,-43.143,-179.042,5.341,148.638
C06302=1232.866,37.021,-43.126,-179.044,5.341,148.639
C06303=1232.871,36.771,-43.110,-179.046,5.341,148.639
C06304=1232.877,36.522,-43.095,-179.049,5.340,148.640
C06305=1232.882,36.273,-43.079,-179.052,5.340,148.641
C06306=1232.887,36.023,-43.063,-179.054,5.339,148.642
C06307=1232.892,35.774,-43.046,-179.057,5.339,148.642
C06308=1232.896,35.524,-43.030,-179.059,5.339,148.643
C06309=1232.901,35.275,-43.014,-179.062,5.338,148.644
C06310=1232.906,35.025,-42.998,-179.064,5.337,148.644
C06311=1232.912,34.776,-42.982,-179.066,5.337,148.645
C06312=1232.917,34.527,-42.966,-179.069,5.336,148.645
C06313=1232.922,34.277,-42.950,-179.072,5.336,148.646
C06314=1232.927,34.027,-42.935,-179.074,5.336,148.647
C06315=1232.931,33.778,-42.918,-179.076,5.335,148.647
C06316=1232.936,33.529,-42.903,-179.079,5.335,148.648
C06317=1232.941,33.279,-42.887,-179.082,5.334,148.649
C06318=1232.946,33.030,-42.871,-179.084,5.334,148.649
C06319=1232.951,32.781,-42.855,-179.087,5.333,148.650
C06320=1232.956,32.530,-42.839,-179.089,5.333,148.651
C06321=1232.961,32.282,-42.823,-179.092,5.333,148.651
C06322=1232.966,32.032,-42.807,-179.094,5.332,148.652
C06323=1232.971,31.782,-42.792,-179.097,5.332,148.653
C06324=1232.976,31.534,-42.776,-179.100,5.331,148.653
C06325=1232.980,31.284,-42.760,-179.102,5.331,148.654
C06326=1232.986,31.034,-42.744,-179.104,5.331,148.655
C06327=1232.991,30.785,-42.728,-179.107,5.330,148.656
C06328=1232.996,30.535,-42.712,-179.110,5.330,148.656
C06329=1233.000,30.286,-42.697,-179.112,5.329,148.657
C06330=1233.006,30.018,-42.680,-179.115,5.329,148.658
C06331=1233.011,29.748,-42.662,-179.118,5.328,148.658
C06332=1233.016,29.480,-42.645,-179.120,5.327,148.659
C06333=1233.022,29.212,-42.628,-179.123,5.327,148.660
C06334=1233.027,28.962,-42.613,-179.125,5.327,148.660
C06335=1233.031,28.712,-42.597,-179.128,5.327,148.661
C06336=1233.037,28.463,-42.582,-179.130,5.326,148.662
C06337=1233.042,28.214,-42.566,-179.133,5.325,148.662
C06338=1233.047,27.963,-42.550,-179.136,5.325,148.663
C06339=1233.052,27.715,-42.534,-179.138,5.325,148.664
C06340=1233.057,27.466,-42.519,-179.140,5.325,148.664
C06341=1233.062,27.215,-42.503,-179.143,5.324,148.665
C06342=1233.067,26.966,-42.487,-179.146,5.324,148.666
C06343=1233.072,26.717,-42.472,-179.148,5.323,148.666
C06344=1233.077,26.468,-42.457,-179.150,5.323,148.667
C06345=1233.082,26.217,-42.441,-179.153,5.323,148.668
C06346=1233.087,25.968,-42.425,-179.156,5.322,148.668
C06347=1233.091,25.720,-42.410,-179.158,5.322,148.669
C06348=1233.096,25.469,-42.394,-179.161,5.321,148.670
C06349=1233.102,25.220,-42.378,-179.163,5.321,148.670
C06350=1233.107,24.971,-42.363,-179.166,5.321,148.671
C06351=1233.112,24.722,-42.348,-179.168,5.320,148.672
C06352=1233.116,24.471,-42.332,-179.171,5.320,148.673
C06353=1233.122,24.222,-42.316,-179.173,5.319,148.673
C06354=1233.126,23.973,-42.301,-179.176,5.319,148.674
C06355=1233.131,23.723,-42.285,-179.178,5.319,148.675
C06356=1233.137,23.473,-42.269,-179.181,5.318,148.675
C06357=1233.141,23.224,-42.254,-179.183,5.318,148.676
C06358=1233.147,22.975,-42.239,-179.186,5.317,148.677
C06359=1233.151,22.725,-42.223,-179.188,5.317,148.677
C06360=1233.156,22.476,-42.208,-179.191,5.317,148.678
C06361=1233.162,22.226,-42.192,-179.193,5.316,148.679
C06362=1233.166,21.977,-42.177,-179.196,5.316,148.679
C06363=1233.171,21.727,-42.161,-179.198,5.316,148.680
C06364=1233.176,21.478,-42.146,-179.201,5.315,148.681
C06365=1233.181,21.229,-42.131,-179.204,5.315,148.681
C06366=1233.186,20.979,-42.115,-179.206,5.314,148.682
C06367=1233.192,20.730,-42.100,-179.209,5.314,148.683
C06368=1233.196,20.480,-42.084,-179.211,5.314,148.683
C06369=1233.201,20.231,-42.069,-179.214,5.314,148.684
C06370=1233.206,19.981,-42.054,-179.216,5.313,148.685
C06371=1233.212,19.732,-42.039,-179.219,5.312,148.685
C06372=1233.216,19.482,-42.023,-179.221,5.313,148.686
C06373=1233.221,19.232,-42.008,-179.224,5.312,148.687
C06374=1233.226,18.983,-41.992,-179.226,5.312,148.688
C06375=1233.231,18.734,-41.977,-179.229,5.311,148.688
C06376=1233.236,18.485,-41.962,-179.231,5.311,148.689
C06377=1233.241,18.235,-41.947,-179.234,5.311,148.690
C06378=1233.246,17.985,-41.931,-179.236,5.310,148.690
C06379=1233.251,17.736,-41.916,-179.239,5.310,148.691
C06380=1233.256,17.486,-41.901,-179.241,5.309,148.692
C06381=1233.261,17.237,-41.886,-179.244,5.309,148.692
C06382=1233.266,16.988,-41.870,-179.246,5.309,148.693
C06383=1233.270,16.738,-41.855,-179.249,5.308,148.694
C06384=1233.276,16.488,-41.840,-179.252,5.308,148.694
C06385=1233.281,16.239,-41.825,-179.254,5.308,148.695
C06386=1233.286,15.989,-41.809,-179.256,5.308,148.696
C06387=1233.291,15.740,-41.795,-179.259,5.307,148.696
C06388=1233.296,15.490,-41.780,-179.262,5.306,148.697
C06389=1233.301,15.241,-41.765,-179.264,5.307,148.698
C06390=1233.306,14.991,-41.749,-179.266,5.306,148.698
C06391=1233.310,14.742,-41.734,-179.269,5.306,148.699
C06392=1233.316,14.492,-41.719,-179.272,5.305,148.700
C06393=1233.321,14.243,-41.704,-179.274,5.305,148.701
C06394=1233.326,13.993,-41.688,-179.276,5.305,148.701
C06395=1233.331,13.744,-41.673,-179.279,5.304,148.702
C06396=1233.336,13.494,-41.658,-179.282,5.304,148.703
C06397=1233.341,13.245,-41.643,-179.284,5.304,148.703
C06398=1233.346,12.995,-41.627,-179.286,5.303,148.704
C06399=1233.351,12.745,-41.613,-179.289,5.303,148.705
C06400=1233.356,12.496,-41.598,-179.292,5.302,148.705
C06401=1233.361,12.247,-41.583,-179.294,5.303,148.706
C06402=1233.366,11.997,-41.568,-179.296,5.302,148.707
C06403=1233.371,11.748,-41.553,-179.299,5.302,148.707
C06404=1233.376,11.499,-41.538,-179.302,5.301,148.708
C06405=1233.381,11.249,-41.523,-179.304,5.301,148.709
C06406=1233.386,11.000,-41.508,-179.306,5.301,148.709
C06407=1233.391,10.751,-41.493,-179.309,5.300,148.710
C06408=1233.397,10.501,-41.478,-179.312,5.300,148.711
C06409=1233.401,10.251,-41.463,-179.314,5.300,148.711
C06410=1233.406,10.001,-41.448,-179.316,5.299,148.712
C06411=1233.411,9.752,-41.433,-179.319,5.299,148.713
C06412=1233.416,9.502,-41.418,-179.322,5.298,148.714
C06413=1233.421,9.253,-41.403,-179.324,5.299,148.714
C06414=1233.426,9.003,-41.388,-179.326,5.298,148.715
C06415=1233.431,8.754,-41.374,-179.329,5.298,148.716
C06416=1233.436,8.505,-41.359,-179.331,5.298,148.716
C06417=1233.441,8.255,-41.344,-179.334,5.297,148.717
C06418=1233.446,8.006,-41.329,-179.336,5.297,148.718
C06419=1233.451,7.756,-41.314,-179.339,5.296,148.718
C06420=1233.456,7.506,-41.299,-179.341,5.296,148.719
C06421=1233.461,7.257,-41.285,-179.344,5.296,148.720
C06422=1233.466,7.008,-41.270,-179.346,5.295,148.720
C06423=1233.472,6.758,-41.255,-179.349,5.295,148.721
C06424=1233.476,6.508,-41.240,-179.351,5.295,148.722
C06425=1233.481,6.259,-41.225,-179.354,5.295,148.722
C06426=1233.486,6.010,-41.210,-179.356,5.294,148.723
C06427=1233.491,5.760,-41.196,-179.359,5.294,148.724
C06428=1233.496,5.511,-41.181,-179.361,5.294,148.725
C06429=1233.501,5.261,-41.166,-179.364,5.293,148.725
C06430=1233.506,5.012,-41.151,-179.367,5.293,148.726
C06431=1233.511,4.762,-41.136,-179.369,5.293,148.727
C06432=1233.516,4.512,-41.122,-179.371,5.292,148.727
C06433=1233.521,4.263,-41.107,-179.374,5.292,148.728
C06434=1233.526,3.994,-41.092,-179.377,5.292,148.729
C06435=1233.532,3.725,-41.075,-179.379,5.292,148.730
C06436=1233.537,3.456,-41.059,-179.382,5.291,148.730
C06437=1233.542,3.187,-41.044,-179.384,5.291,148.731
C06438=1233.548,2.937,-41.029,-179.387,5.290,148.732
C06439=1233.553,2.688,-41.015,-179.390,5.290,148.732
C06440=1233.558,2.439,-41.000,-179.392,5.290,148.733
C06441=1233.563,2.189,-40.985,-179.394,5.290,148.734
C06442=1233.567,1.939,-40.971,-179.398,5.289,148.735
C06443=1233.573,1.690,-40.956,-179.400,5.290,148.735
C06444=1233.578,1.440,-40.941,-179.402,5.289,148.736
C06445=1233.583,1.191,-40.927,-179.405,5.289,148.737
C06446=1233.588,0.942,-40.912,-179.408,5.288,148.737
C06447=1233.593,0.692,-40.898,-179.410,5.288,148.738
C06448=1233.598,0.443,-40.884,-179.412,5.288,148.739
C06449=1233.603,0.193,-40.868,-179.415,5.287,148.739
C06450=1233.608,-0.057,-40.854,-179.417,5.288,148.740
C06451=1233.613,-0.306,-40.840,-179.420,5.287,148.741
C06452=1233.618,-0.556,-40.825,-179.422,5.287,148.741
C06453=1233.623,-0.805,-40.810,-179.424,5.287,148.742
C06454=1233.628,-1.055,-40.796,-179.427,5.286,148.743
C06455=1233.633,-1.304,-40.782,-179.430,5.286,148.744
C06456=1233.638,-1.554,-40.768,-179.432,5.285,148.744
C06457=1233.644,-1.803,-40.752,-179.435,5.286,148.745
C06458=1233.649,-2.053,-40.738,-179.437,5.285,148.746
C06459=1233.654,-2.302,-40.724,-179.440,5.285,148.746
C06460=1233.659,-2.552,-40.709,-179.442,5.285,148.747
C06461=1233.663,-2.801,-40.694,-179.445,5.284,148.748
C06462=1233.668,-3.051,-40.680,-179.447,5.284,148.748
C06463=1233.673,-3.301,-40.666,-179.449,5.284,148.749
C06464=1233.678,-3.550,-40.652,-179.452,5.284,148.750
C06465=1233.683,-3.800,-40.637,-179.455,5.283,148.750
C06466=1233.689,-4.049,-40.623,-179.457,5.283,148.751
C06467=1233.693,-4.298,-40.608,-179.459,5.283,148.752
C06468=1233.698,-4.548,-40.594,-179.462,5.282,148.753
C06469=1233.703,-4.797,-40.580,-179.465,5.282,148.753
C06470=1233.708,-5.047,-40.566,-179.467,5.282,148.754
C06471=1233.714,-5.297,-40.551,-179.469,5.281,148.755
C06472=1233.719,-5.547,-40.536,-179.473,5.281,148.756
C06473=1233.724,-5.796,-40.523,-179.475,5.282,148.756
C06474=1233.729,-6.046,-40.508,-179.477,5.281,148.757
C06475=1233.734,-6.295,-40.494,-179.480,5.281,148.758
C06476=1233.739,-6.544,-40.479,-179.482,5.281,148.758
C06477=1233.744,-6.794,-40.465,-179.485,5.280,148.759
C06478=1233.749,-7.044,-40.450,-179.487,5.280,148.760
C06479=1233.754,-7.293,-40.437,-179.489,5.280,148.760
C06480=1233.759,-7.542,-40.423,-179.492,5.280,148.761
C06481=1233.763,-7.792,-40.409,-179.495,5.279,148.762
C06482=1233.768,-8.042,-40.394,-179.497,5.279,148.762
C06483=1233.773,-8.291,-40.380,-179.499,5.279,148.763
C06484=1233.779,-8.540,-40.366,-179.502,5.278,148.764
C06485=1233.784,-8.790,-40.352,-179.504,5.279,148.765
C06486=1233.789,-9.040,-40.338,-179.507,5.278,148.765
C06487=1233.794,-9.290,-40.323,-179.509,5.277,148.766
C06488=1233.799,-9.539,-40.309,-179.512,5.278,148.767
C06489=1233.804,-9.788,-40.295,-179.514,5.277,148.767
C06490=1233.809,-10.038,-40.281,-179.517,5.277,148.768
C06491=1233.814,-10.288,-40.267,-179.519,5.277,148.769
C06492=1233.819,-10.537,-40.252,-179.522,5.276,148.769
C06493=1233.825,-10.786,-40.238,-179.524,5.276,148.770
C06494=1233.830,-11.036,-40.224,-179.526,5.276,148.771
C06495=1233.835,-11.286,-40.210,-179.530,5.276,148.772
C06496=1233.839,-11.535,-40.196,-179.532,5.276,148.772
C06497=1233.844,-11.785,-40.182,-179.534,5.276,148.773
C06498=1233.849,-12.034,-40.168,-179.537,5.275,148.774
C06499=1233.855,-12.284,-40.154,-179.540,5.275,148.774
C06500=1233.860,-12.534,-40.140,-179.542,5.275,148.775
C06501=1233.865,-12.784,-40.126,-179.544,5.275,148.776
C06502=1233.870,-13.033,-40.112,-179.547,5.274,148.777
C06503=1233.875,-13.282,-40.098,-179.549,5.274,148.777
C06504=1233.879,-13.532,-40.084,-179.552,5.274,148.778
C06505=1233.885,-13.781,-40.070,-179.554,5.273,148.779
C06506=1233.890,-14.031,-40.056,-179.556,5.274,148.779
C06507=1233.895,-14.281,-40.042,-179.559,5.273,148.780
C06508=1233.900,-14.531,-40.028,-179.562,5.273,148.781
C06509=1233.906,-14.780,-40.014,-179.564,5.273,148.781
C06510=1233.910,-15.029,-40.000,-179.566,5.272,148.782
C06511=1233.915,-15.279,-39.986,-179.569,5.272,148.783
C06512=1233.920,-15.528,-39.972,-179.571,5.272,148.783
C06513=1233.926,-15.778,-39.959,-179.574,5.272,148.784
C06514=1233.931,-16.028,-39.944,-179.577,5.271,148.785
C06515=1233.935,-16.277,-39.931,-179.579,5.271,148.786
C06516=1233.940,-16.526,-39.917,-179.582,5.271,148.786
C06517=1233.945,-16.776,-39.902,-179.584,5.272,148.787
C06518=1233.950,-17.026,-39.889,-179.586,5.271,148.788
C06519=1233.956,-17.275,-39.875,-179.589,5.271,148.789
C06520=1233.960,-17.525,-39.861,-179.591,5.271,148.789
C06521=1233.965,-17.774,-39.847,-179.594,5.270,148.790
C06522=1233.971,-18.024,-39.834,-179.597,5.270,148.791
C06523=1233.976,-18.274,-39.820,-179.599,5.270,148.791
C06524=1233.980,-18.523,-39.806,-179.601,5.270,148.792
C06525=1233.986,-18.773,-39.793,-179.604,5.269,148.793
C06526=1233.991,-19.022,-39.778,-179.606,5.269,148.793
C06527=1233.996,-19.272,-39.764,-179.609,5.269,148.794
C06528=1234.001,-19.521,-39.751,-179.611,5.268,148.795
C06529=1234.006,-19.771,-39.737,-179.613,5.269,148.796
C06530=1234.012,-20.020,-39.723,-179.616,5.268,148.796
C06531=1234.017,-20.270,-39.709,-179.618,5.268,148.797
C06532=1234.021,-20.520,-39.696,-179.621,5.268,148.798
C06533=1234.027,-20.769,-39.682,-179.623,5.267,148.798
C06534=1234.032,-21.019,-39.668,-179.626,5.268,148.799
C06535=1234.036,-21.269,-39.655,-179.629,5.268,148.800
C06536=1234.042,-21.518,-39.641,-179.631,5.267,148.801
C06537=1234.047,-21.768,-39.627,-179.633,5.267,148.801
C06538=1234.052,-22.037,-39.612,-179.636,5.267,148.802
C06539=1234.058,-22.306,-39.598,-179.639,5.266,148.803
C06540=1234.063,-22.575,-39.583,-179.642,5.266,148.804
C06541=1234.069,-22.845,-39.568,-179.644,5.266,148.804
C06542=1234.074,-23.094,-39.554,-179.647,5.266,148.805
C06543=1234.079,-23.344,-39.542,-179.649,5.265,148.806
C06544=1234.084,-23.593,-39.527,-179.651,5.266,148.806
C06545=1234.089,-23.843,-39.514,-179.654,5.265,148.807
C06546=1234.094,-24.092,-39.500,-179.656,5.266,148.808
C06547=1234.100,-24.342,-39.487,-179.659,5.265,148.808
C06548=1234.104,-24.591,-39.474,-179.661,5.264,148.809
C06549=1234.109,-24.841,-39.459,-179.664,5.265,148.810
C06550=1234.115,-25.091,-39.446,-179.666,5.264,148.811
C06551=1234.119,-25.340,-39.432,-179.669,5.264,148.811
C06552=1234.125,-25.590,-39.419,-179.671,5.264,148.812
C06553=1234.129,-25.839,-39.405,-179.674,5.264,148.813
C06554=1234.135,-26.089,-39.392,-179.676,5.264,148.814
C06555=1234.140,-26.338,-39.378,-179.679,5.264,148.814
C06556=1234.144,-26.589,-39.365,-179.682,5.263,148.815
C06557=1234.150,-26.838,-39.351,-179.684,5.264,148.816
C06558=1234.154,-27.088,-39.338,-179.686,5.263,148.816
C06559=1234.160,-27.337,-39.325,-179.689,5.263,148.817
C06560=1234.164,-27.587,-39.311,-179.691,5.263,148.818
C06561=1234.170,-27.836,-39.298,-179.694,5.262,148.818
C06562=1234.174,-28.086,-39.284,-179.696,5.263,148.819
C06563=1234.180,-28.335,-39.271,-179.698,5.262,148.820
C06564=1234.185,-28.585,-39.258,-179.701,5.262,148.821
C06565=1234.190,-28.834,-39.244,-179.703,5.262,148.821
C06566=1234.196,-29.085,-39.231,-179.706,5.261,148.822
C06567=1234.200,-29.333,-39.217,-179.708,5.262,148.823
C06568=1234.206,-29.584,-39.204,-179.711,5.261,148.823
C06569=1234.211,-29.832,-39.191,-179.713,5.261,148.824
C06570=1234.216,-30.083,-39.177,-179.716,5.261,148.825
C06571=1234.221,-30.332,-39.164,-179.718,5.261,148.826
C06572=1234.226,-30.582,-39.150,-179.721,5.260,148.826
C06573=1234.231,-30.831,-39.138,-179.723,5.261,148.827
C06574=1234.236,-31.081,-39.124,-179.726,5.260,148.828
C06575=1234.241,-31.330,-39.111,-179.728,5.260,148.828
C06576=1234.246,-31.580,-39.098,-179.731,5.260,148.829
C06577=1234.251,-31.830,-39.085,-179.733,5.259,148.830
C06578=1234.256,-32.079,-39.071,-179.735,5.260,148.831
C06579=1234.262,-32.329,-39.058,-179.738,5.259,148.831
C06580=1234.266,-32.579,-39.045,-179.740,5.260,148.832
C06581=1234.272,-32.828,-39.031,-179.743,5.259,148.833
C06582=1234.276,-33.078,-39.018,-179.745,5.259,148.833
C06583=1234.282,-33.327,-39.005,-179.748,5.259,148.834
C06584=1234.286,-33.577,-38.991,-179.750,5.258,148.835
C06585=1234.291,-33.826,-38.978,-179.752,5.259,148.835
C06586=1234.297,-34.076,-38.965,-179.755,5.259,148.836
C06587=1234.302,-34.326,-38.952,-179.758,5.258,148.837
C06588=1234.307,-34.575,-38.938,-179.760,5.258,148.838
C06589=1234.312,-34.825,-38.925,-179.763,5.258,148.838
C06590=1234.318,-35.074,-38.912,-179.765,5.258,148.839
C06591=1234.322,-35.324,-38.899,-179.768,5.258,148.840
C06592=1234.327,-35.574,-38.887,-179.770,5.257,148.841
C06593=1234.333,-35.823,-38.873,-179.772,5.257,148.841
C06594=1234.337,-36.073,-38.860,-179.775,5.257,148.842
C06595=1234.343,-36.322,-38.847,-179.777,5.257,148.843
C06596=1234.348,-36.572,-38.833,-179.780,5.257,148.843
C06597=1234.353,-36.822,-38.821,-179.782,5.257,148.844
C06598=1234.358,-37.071,-38.807,-179.784,5.257,148.845
C06599=1234.363,-37.321,-38.794,-179.787,5.256,148.845
C06600=1234.368,-37.570,-38.781,-179.789,5.256,148.846
C06601=1234.373,-37.820,-38.768,-179.792,5.256,148.847
C06602=1234.379,-38.070,-38.755,-179.794,5.256,148.848
C06603=1234.384,-38.319,-38.743,-179.797,5.256,148.849
C06604=1234.389,-38.569,-38.729,-179.800,5.256,148.849
C06605=1234.394,-38.818,-38.716,-179.802,5.256,148.850
C06606=1234.398,-39.068,-38.703,-179.805,5.255,148.851
C06607=1234.404,-39.318,-38.690,-179.807,5.256,148.851
C06608=1234.409,-39.567,-38.677,-179.809,5.255,148.852
C06609=1234.414,-39.817,-38.664,-179.812,5.255,148.853
C06610=1234.419,-40.066,-38.651,-179.814,5.255,148.853
C06611=1234.425,-40.316,-38.638,-179.817,5.255,148.854
C06612=1234.429,-40.566,-38.625,-179.819,5.255,148.855
C06613=1234.434,-40.815,-38.613,-179.821,5.254,148.856
C06614=1234.440,-41.065,-38.599,-179.824,5.255,148.856
C06615=1234.445,-41.315,-38.586,-179.826,5.254,148.857
C06616=1234.450,-41.564,-38.574,-179.829,5.254,148.858
C06617=1234.455,-41.814,-38.561,-179.831,5.254,148.858
C06618=1234.460,-42.064,-38.548,-179.834,5.253,148.859
C06619=1234.465,-42.313,-38.535,-179.836,5.254,148.860
C06620=1234.471,-42.563,-38.523,-179.839,5.254,148.861
C06621=1234.475,-42.813,-38.510,-179.841,5.254,148.861
C06622=1234.481,-43.062,-38.496,-179.844,5.254,148.862
C06623=1234.486,-43.312,-38.484,-179.846,5.253,148.863
C06624=1234.491,-43.562,-38.471,-179.848,5.253,148.863
C06625=1234.496,-43.811,-38.458,-179.851,5.253,148.864
C06626=1234.501,-44.060,-38.446,-179.853,5.253,148.865
C06627=1234.506,-44.311,-38.432,-179.856,5.253,148.866
C06628=1234.511,-44.560,-38.419,-179.858,5.253,148.866
C06629=1234.516,-44.809,-38.407,-179.861,5.252,148.867
C06630=1234.521,-45.059,-38.394,-179.863,5.252,148.868
C06631=1234.526,-45.308,-38.381,-179.865,5.252,148.868
C06632=1234.532,-45.558,-38.368,-179.868,5.252,148.869
C06633=1234.537,-45.807,-38.355,-179.870,5.252,148.870
C06634=1234.541,-46.057,-38.343,-179.873,5.252,148.870
C06635=1234.547,-46.307,-38.330,-179.875,5.252,148.871
C06636=1234.552,-46.556,-38.317,-179.878,5.252,148.872
C06637=1234.556,-46.806,-38.304,-179.881,5.251,148.873
C06638=1234.562,-47.056,-38.292,-179.883,5.252,148.874
C06639=1234.568,-47.306,-38.279,-179.885,5.251,148.874
C06640=1234.573,-47.555,-38.267,-179.887,5.251,148.875
C06641=1234.577,-47.805,-38.254,-179.890,5.251,148.876
C06642=1234.583,-48.074,-38.240,-179.893,5.251,148.876
C06643=1234.589,-48.344,-38.226,-179.895,5.251,148.877
C06644=1234.594,-48.614,-38.212,-179.898,5.251,148.878
C06645=1234.600,-48.884,-38.199,-179.901,5.250,148.879
C06646=1234.605,-49.133,-38.187,-179.903,5.251,148.879
C06647=1234.610,-49.383,-38.174,-179.905,5.250,148.880
C06648=1234.615,-49.632,-38.161,-179.908,5.250,148.881
C06649=1234.620,-49.882,-38.148,-179.910,5.250,148.881
C06650=1234.625,-50.132,-38.137,-179.912,5.250,148.882
C06651=1234.630,-50.382,-38.124,-179.915,5.250,148.883
C06652=1234.635,-50.631,-38.111,-179.918,5.250,148.884
C06653=1234.640,-50.880,-38.098,-179.920,5.250,148.885
C06654=1234.645,-51.130,-38.086,-179.923,5.249,148.885
C06655=1234.651,-51.380,-38.074,-179.925,5.250,148.886
C06656=1234.655,-51.630,-38.061,-179.928,5.249,148.887
C06657=1234.660,-51.879,-38.048,-179.930,5.250,148.887
C06658=1234.666,-52.129,-38.036,-179.932,5.249,148.888
C06659=1234.671,-52.378,-38.024,-179.934,5.249,148.889
C06660=1234.676,-52.627,-38.011,-179.937,5.249,148.889
C06661=1234.681,-52.878,-37.998,-179.939,5.249,148.890
C06662=1234.687,-53.128,-37.986,-179.942,5.249,148.891
C06663=1234.692,-53.377,-37.973,-179.945,5.248,148.892
C06664=1234.697,-53.626,-37.961,-179.947,5.249,148.892
C06665=1234.702,-53.876,-37.949,-179.949,5.248,148.893
C06666=1234.707,-54.126,-37.936,-179.951,5.248,148.894
C06667=1234.712,-54.376,-37.923,-179.954,5.248,148.894
C06668=1234.718,-54.626,-37.911,-179.956,5.248,148.895
C06669=1234.722,-54.875,-37.899,-179.959,5.248,148.896
C06670=1234.727,-55.124,-37.887,-179.961,5.249,148.897
C06671=1234.733,-55.374,-37.875,-179.964,5.248,148.897
C06672=1234.737,-55.624,-37.862,-179.966,5.248,148.898
C06673=1234.742,-55.873,-37.849,-179.969,5.248,148.899
C06674=1234.748,-56.123,-37.837,-179.971,5.247,148.900
C06675=1234.753,-56.372,-37.825,-179.974,5.248,148.900
C06676=1234.758,-56.622,-37.812,-179.976,5.247,148.901
C06677=1234.763,-56.872,-37.800,-179.978,5.248,148.902
C06678=1234.768,-57.121,-37.788,-179.981,5.247,148.902
C06679=1234.773,-57.372,-37.775,-179.983,5.247,148.903
C06680=1234.778,-57.621,-37.763,-179.986,5.247,148.904
C06681=1234.784,-57.871,-37.751,-179.988,5.247,148.904
C06682=1234.789,-58.120,-37.738,-179.991,5.247,148.905
C06683=1234.794,-58.370,-37.726,-179.993,5.247,148.906
C06684=1234.799,-58.619,-37.714,-179.995,5.247,148.907
C06685=1234.804,-58.868,-37.702,-179.998,5.246,148.907
C06686=1234.809,-59.118,-37.690,180.000,5.246,148.908
C06687=1234.814,-59.368,-37.677,179.997,5.246,148.909
C06688=1234.819,-59.618,-37.665,179.995,5.247,148.910
C06689=1234.824,-59.868,-37.652,179.992,5.246,148.910
C06690=1234.830,-60.118,-37.641,179.990,5.247,148.911
C06691=1234.835,-60.367,-37.628,179.987,5.246,148.912
C06692=1234.840,-60.617,-37.616,179.985,5.246,148.912
C06693=1234.845,-60.866,-37.603,179.983,5.246,148.913
C06694=1234.850,-61.116,-37.592,179.980,5.246,148.914
C06695=1234.855,-61.365,-37.580,179.978,5.246,148.915
C06696=1234.861,-61.615,-37.568,179.976,5.246,148.915
C06697=1234.866,-61.864,-37.555,179.973,5.246,148.916
C06698=1234.871,-62.114,-37.543,179.971,5.246,148.917
C06699=1234.876,-62.364,-37.531,179.968,5.245,148.917
C06700=1234.881,-62.613,-37.519,179.966,5.245,148.918
C06701=1234.886,-62.864,-37.507,179.964,5.245,148.919
C06702=1234.891,-63.113,-37.494,179.961,5.245,148.920
C06703=1234.896,-63.363,-37.483,179.959,5.245,148.920
C06704=1234.902,-63.612,-37.470,179.956,5.245,148.921
C06705=1234.906,-63.862,-37.459,179.954,5.245,148.922
C06706=1234.912,-64.112,-37.447,179.951,5.245,148.922
C06707=1234.917,-64.361,-37.434,179.949,5.245,148.923
C06708=1234.922,-64.611,-37.422,179.946,5.245,148.924
C06709=1234.927,-64.861,-37.410,179.944,5.245,148.925
C06710=1234.932,-65.110,-37.398,179.941,5.245,148.925
C06711=1234.937,-65.360,-37.387,179.939,5.245,148.926
C06712=1234.943,-65.609,-37.374,179.937,5.244,148.927
C06713=1234.948,-65.859,-37.362,179.934,5.245,148.928
C06714=1234.953,-66.109,-37.351,179.932,5.244,148.928
C06715=1234.958,-66.358,-37.338,179.930,5.245,148.929
C06716=1234.963,-66.608,-37.326,179.927,5.244,148.930
C06717=1234.969,-66.858,-37.314,179.925,5.244,148.930
C06718=1234.973,-67.107,-37.302,179.922,5.244,148.931
C06719=1234.979,-67.357,-37.291,179.920,5.244,148.932
C06720=1234.984,-67.607,-37.279,179.918,5.244,148.932
C06721=1234.989,-67.857,-37.267,179.915,5.243,148.933
C06722=1234.994,-68.106,-37.255,179.913,5.244,148.934
C06723=1234.999,-68.356,-37.243,179.910,5.243,148.935
C06724=1235.005,-68.606,-37.231,179.908,5.244,148.935
C06725=1235.009,-68.855,-37.219,179.905,5.243,148.936
C06726=1235.014,-69.105,-37.207,179.903,5.243,148.937
C06727=1235.020,-69.355,-37.195,179.901,5.243,148.937
C06728=1235.025,-69.605,-37.183,179.899,5.243,148.938
C06729=1235.030,-69.854,-37.172,179.896,5.243,148.939
C06730=1235.035,-70.104,-37.159,179.894,5.243,148.940
C06731=1235.041,-70.354,-37.148,179.891,5.243,148.940
C06732=1235.046,-70.603,-37.137,179.888,5.243,148.941
C06733=1235.051,-70.852,-37.125,179.886,5.243,148.942
C06734=1235.056,-71.102,-37.112,179.884,5.243,148.943
C06735=1235.061,-71.351,-37.101,179.881,5.243,148.943
C06736=1235.067,-71.601,-37.089,179.879,5.243,148.944
C06737=1235.072,-71.851,-37.077,179.876,5.243,148.945
C06738=1235.077,-72.101,-37.066,179.874,5.243,148.945
C06739=1235.082,-72.351,-37.054,179.872,5.243,148.946
C06740=1235.086,-72.600,-37.042,179.869,5.243,148.947
C06741=1235.092,-72.850,-37.030,179.867,5.242,148.948
C06742=1235.097,-73.100,-37.018,179.865,5.243,148.948
C06743=1235.102,-73.349,-37.007,179.862,5.242,148.949
C06744=1235.107,-73.599,-36.995,179.860,5.243,148.950
C06745=1235.113,-73.849,-36.983,179.857,5.242,148.950
C06746=1235.119,-74.119,-36.970,179.855,5.242,148.951
C06747=1235.124,-74.389,-36.958,179.852,5.242,148.952
C06748=1235.130,-74.660,-36.946,179.849,5.242,148.953
C06749=1235.136,-74.930,-36.933,179.847,5.242,148.953
C06750=1235.140,-75.180,-36.921,179.845,5.242,148.954
C06751=1235.146,-75.429,-36.909,179.842,5.242,148.955
C06752=1235.150,-75.679,-36.898,179.840,5.242,148.956
C06753=1235.156,-75.928,-36.887,179.838,5.242,148.956
C06754=1235.161,-76.178,-36.875,179.835,5.242,148.957
C06755=1235.167,-76.428,-36.863,179.833,5.242,148.958
C06756=1235.172,-76.677,-36.851,179.830,5.241,148.958
C06757=1235.176,-76.927,-36.840,179.828,5.242,148.959
C06758=1235.182,-77.177,-36.828,179.826,5.241,148.960
C06759=1235.187,-77.426,-36.816,179.823,5.242,148.961
C06760=1235.193,-77.676,-36.805,179.820,5.242,148.962
C06761=1235.197,-77.925,-36.794,179.818,5.242,148.962
C06762=1235.203,-78.175,-36.782,179.815,5.241,148.963
C06763=1235.207,-78.425,-36.770,179.813,5.242,148.964
C06764=1235.213,-78.675,-36.759,179.811,5.241,148.964
C06765=1235.217,-78.924,-36.747,179.809,5.242,148.965
C06766=1235.223,-79.174,-36.735,179.806,5.241,148.966
C06767=1235.228,-79.424,-36.725,179.804,5.242,148.966
C06768=1235.234,-79.674,-36.713,179.801,5.241,148.967
C06769=1235.239,-79.923,-36.702,179.799,5.241,148.968
C06770=1235.244,-80.173,-36.690,179.796,5.241,148.969
C06771=1235.249,-80.423,-36.679,179.794,5.241,148.969
C06772=1235.255,-80.672,-36.667,179.792,5.241,148.970
C06773=1235.259,-80.922,-36.656,179.790,5.241,148.971
C06774=1235.264,-81.171,-36.645,179.787,5.241,148.971
C06775=1235.270,-81.421,-36.633,179.785,5.241,148.972
C06776=1235.274,-81.671,-36.622,179.782,5.241,148.973
C06777=1235.280,-81.920,-36.610,179.780,5.241,148.974
C06778=1235.285,-82.170,-36.599,179.777,5.240,148.974
C06779=1235.291,-82.420,-36.588,179.775,5.241,148.975
C06780=1235.295,-82.670,-36.576,179.773,5.240,148.976
C06781=1235.300,-82.920,-36.565,179.771,5.241,148.976
C06782=1235.306,-83.169,-36.553,179.768,5.240,148.977
C06783=1235.311,-83.419,-36.542,179.766,5.241,148.978
C06784=1235.316,-83.668,-36.530,179.763,5.240,148.979
C06785=1235.321,-83.918,-36.519,179.761,5.240,148.979
C06786=1235.326,-84.168,-36.508,179.758,5.240,148.980
C06787=1235.332,-84.418,-36.497,179.756,5.240,148.981
C06788=1235.337,-84.667,-36.486,179.754,5.240,148.981
C06789=1235.342,-84.917,-36.474,179.751,5.240,148.982
C06790=1235.347,-85.167,-36.462,179.749,5.240,148.983
C06791=1235.352,-85.416,-36.452,179.747,5.240,148.984
C06792=1235.358,-85.666,-36.440,179.744,5.240,148.984
C06793=1235.363,-85.916,-36.429,179.742,5.240,148.985
C06794=1235.367,-86.166,-36.418,179.739,5.240,148.986
C06795=1235.373,-86.415,-36.406,179.737,5.240,148.986
C06796=1235.378,-86.665,-36.396,179.734,5.239,148.987
C06797=1235.383,-86.915,-36.384,179.732,5.240,148.988
C06798=1235.389,-87.164,-36.373,179.730,5.239,148.988
C06799=1235.394,-87.413,-36.362,179.728,5.240,148.989
C06800=1235.399,-87.664,-36.351,179.725,5.239,148.990
C06801=1235.404,-87.914,-36.339,179.723,5.240,148.991
C06802=1235.409,-88.163,-36.328,179.720,5.239,148.991
C06803=1235.414,-88.412,-36.317,179.718,5.239,148.992
C06804=1235.420,-88.663,-36.306,179.715,5.239,148.993
C06805=1235.425,-88.912,-36.295,179.713,5.239,148.993
C06806=1235.430,-89.161,-36.284,179.711,5.240,148.994
C06807=1235.436,-89.412,-36.272,179.709,5.239,148.995
C06808=1235.440,-89.661,-36.261,179.706,5.240,148.996
C06809=1235.446,-89.910,-36.250,179.704,5.239,148.996
C06810=1235.451,-90.161,-36.240,179.702,5.239,148.997
C06811=1235.456,-90.411,-36.228,179.699,5.239,148.998
C06812=1235.461,-90.660,-36.217,179.697,5.239,148.998
C06813=1235.466,-90.910,-36.206,179.694,5.239,148.999
C06814=1235.471,-91.159,-36.195,179.692,5.239,149.000
C06815=1235.477,-91.409,-36.183,179.690,5.239,149.001
C06816=1235.482,-91.659,-36.173,179.687,5.239,149.001
C06817=1235.487,-91.909,-36.162,179.685,5.239,149.002
C06818=1235.492,-92.158,-36.151,179.683,5.239,149.003
C06819=1235.498,-92.408,-36.139,179.680,5.239,149.003
C06820=1235.502,-92.658,-36.128,179.678,5.239,149.004
C06821=1235.508,-92.907,-36.118,179.675,5.239,149.005
C06822=1235.513,-93.157,-36.107,179.673,5.239,149.006
C06823=1235.518,-93.407,-36.096,179.670,5.238,149.006
C06824=1235.524,-93.656,-36.085,179.668,5.239,149.007
C06825=1235.529,-93.907,-36.074,179.666,5.238,149.008
C06826=1235.534,-94.155,-36.063,179.664,5.239,149.008
C06827=1235.539,-94.405,-36.052,179.661,5.238,149.009
C06828=1235.544,-94.655,-36.041,179.659,5.239,149.010
C06829=1235.550,-94.905,-36.030,179.657,5.239,149.011
C06830=1235.555,-95.155,-36.019,179.654,5.238,149.011
C06831=1235.559,-95.404,-36.008,179.652,5.239,149.012
C06832=1235.565,-95.654,-35.998,179.649,5.238,149.013
C06833=1235.570,-95.904,-35.986,179.647,5.239,149.013
C06834=1235.576,-96.153,-35.975,179.645,5.238,149.014
C06835=1235.581,-96.403,-35.964,179.642,5.239,149.015
C06836=1235.586,-96.653,-35.954,179.640,5.238,149.016
C06837=1235.591,-96.902,-35.943,179.638,5.239,149.016
C06838=1235.596,-97.152,-35.932,179.635,5.238,149.017
C06839=1235.601,-97.401,-35.921,179.633,5.238,149.018
C06840=1235.606,-97.652,-35.911,179.630,5.238,149.018
C06841=1235.612,-97.902,-35.899,179.628,5.238,149.019
C06842=1235.617,-98.151,-35.889,179.625,5.238,149.020
C06843=1235.622,-98.401,-35.878,179.623,5.238,149.021
C06844=1235.628,-98.650,-35.867,179.621,5.238,149.021
C06845=1235.633,-98.901,-35.856,179.619,5.238,149.022
C06846=1235.638,-99.149,-35.846,179.616,5.238,149.023
C06847=1235.643,-99.400,-35.835,179.614,5.238,149.023
C06848=1235.648,-99.649,-35.824,179.612,5.238,149.024
C06849=1235.653,-99.899,-35.813,179.609,5.238,149.025
C06850=1235.659,-100.170,-35.801,179.607,5.238,149.026
C06851=1235.665,-100.441,-35.790,179.604,5.238,149.026
C06852=1235.670,-100.711,-35.778,179.601,5.238,149.027
C06853=1235.676,-100.983,-35.767,179.599,5.238,149.028
C06854=1235.681,-101.232,-35.756,179.596,5.238,149.029
C06855=1235.686,-101.482,-35.745,179.594,5.238,149.029
C06856=1235.691,-101.732,-35.735,179.592,5.238,149.030
C06857=1235.697,-101.981,-35.724,179.589,5.238,149.031
C06858=1235.702,-102.232,-35.713,179.587,5.238,149.031
C06859=1235.707,-102.481,-35.703,179.585,5.238,149.032
C06860=1235.712,-102.731,-35.692,179.583,5.238,149.033
C06861=1235.718,-102.980,-35.682,179.580,5.238,149.034
C06862=1235.723,-103.231,-35.671,179.578,5.238,149.034
C06863=1235.728,-103.479,-35.660,179.575,5.238,149.035
C06864=1235.733,-103.730,-35.649,179.573,5.238,149.036
C06865=1235.738,-103.979,-35.639,179.570,5.238,149.036
C06866=1235.743,-104.229,-35.628,179.568,5.238,149.037
C06867=1235.749,-104.478,-35.618,179.566,5.238,149.038
C06868=1235.754,-104.729,-35.607,179.564,5.238,149.039
C06869=1235.759,-104.978,-35.597,179.561,5.237,149.039
C06870=1235.764,-105.228,-35.586,179.559,5.237,149.040
C06871=1235.770,-105.477,-35.575,179.557,5.237,149.041
C06872=1235.775,-105.728,-35.565,179.554,5.237,149.041
C06873=1235.780,-105.977,-35.555,179.552,5.238,149.042
C06874=1235.785,-106.227,-35.543,179.550,5.237,149.043
C06875=1235.791,-106.476,-35.533,179.548,5.238,149.043
C06876=1235.796,-106.727,-35.523,179.545,5.237,149.044
C06877=1235.801,-106.976,-35.512,179.543,5.238,149.045
C06878=1235.807,-107.226,-35.502,179.540,5.237,149.046
C06879=1235.811,-107.475,-35.491,179.538,5.237,149.046
C06880=1235.816,-107.725,-35.481,179.535,5.237,149.047
C06881=1235.821,-107.975,-35.471,179.533,5.237,149.048
C06882=1235.827,-108.224,-35.461,179.531,5.237,149.048
C06883=1235.832,-108.475,-35.450,179.529,5.237,149.049
C06884=1235.837,-108.723,-35.439,179.526,5.238,149.050
C06885=1235.842,-108.974,-35.428,179.524,5.237,149.051
C06886=1235.848,-109.223,-35.418,179.522,5.238,149.051
C06887=1235.853,-109.473,-35.408,179.519,5.237,149.052
C06888=1235.858,-109.723,-35.397,179.517,5.238,149.053
C06889=1235.864,-109.973,-35.387,179.514,5.237,149.053
C06890=1235.868,-110.223,-35.377,179.512,5.237,149.054
C06891=1235.874,-110.472,-35.367,179.509,5.237,149.055
C06892=1235.878,-110.722,-35.356,179.507,5.237,149.056
C06893=1235.884,-110.971,-35.346,179.505,5.237,149.056
C06894=1235.890,-111.221,-35.335,179.503,5.237,149.057
C06895=1235.895,-111.471,-35.325,179.501,5.237,149.057
C06896=1235.900,-111.721,-35.315,179.498,5.237,149.058
C06897=1235.905,-111.971,-35.304,179.496,5.237,149.059
C06898=1235.910,-112.220,-35.294,179.493,5.237,149.060
C06899=1235.916,-112.470,-35.284,179.491,5.237,149.060
C06900=1235.921,-112.720,-35.274,179.489,5.237,149.061
C06901=1235.926,-112.969,-35.263,179.487,5.237,149.062
C06902=1235.931,-113.220,-35.253,179.484,5.237,149.062
C06903=1235.937,-113.469,-35.243,179.482,5.237,149.063
C06904=1235.942,-113.718,-35.233,179.479,5.237,149.064
C06905=1235.947,-113.969,-35.222,179.477,5.237,149.065
C06906=1235.952,-114.218,-35.212,179.475,5.237,149.065
C06907=1235.958,-114.468,-35.202,179.472,5.237,149.066
C06908=1235.963,-114.718,-35.191,179.470,5.237,149.067
C06909=1235.968,-114.967,-35.182,179.468,5.237,149.067
C06910=1235.973,-115.217,-35.172,179.466,5.237,149.068
C06911=1235.978,-115.467,-35.161,179.463,5.236,149.069
C06912=1235.984,-115.717,-35.151,179.461,5.237,149.069
C06913=1235.988,-115.966,-35.141,179.458,5.236,149.070
C06914=1235.994,-116.216,-35.131,179.456,5.237,149.071
C06915=1235.999,-116.466,-35.120,179.454,5.237,149.072
C06916=1236.004,-116.716,-35.110,179.452,5.237,149.072
C06917=1236.010,-116.965,-35.100,179.450,5.237,149.073
C06918=1236.015,-117.215,-35.090,179.447,5.237,149.074
C06919=1236.020,-117.465,-35.079,179.445,5.237,149.074
C06920=1236.026,-117.714,-35.069,179.442,5.236,149.075
C06921=1236.030,-117.964,-35.060,179.440,5.237,149.076
C06922=1236.035,-118.214,-35.049,179.437,5.236,149.077
C06923=1236.041,-118.464,-35.040,179.435,5.237,149.077
C06924=1236.047,-118.714,-35.029,179.434,5.237,149.078
C06925=1236.052,-118.963,-35.020,179.431,5.236,149.078
C06926=1236.057,-119.213,-35.009,179.429,5.237,149.079
C06927=1236.062,-119.463,-34.999,179.426,5.236,149.080
C06928=1236.067,-119.712,-34.989,179.424,5.237,149.081
C06929=1236.072,-119.962,-34.979,179.421,5.236,149.081
C06930=1236.078,-120.212,-34.969,179.419,5.237,149.082
C06931=1236.083,-120.461,-34.960,179.417,5.236,149.083
C06932=1236.088,-120.712,-34.949,179.414,5.236,149.083
C06933=1236.094,-120.961,-34.939,179.412,5.237,149.084
C06934=1236.098,-121.210,-34.929,179.410,5.236,149.085
C06935=1236.104,-121.460,-34.919,179.408,5.237,149.086
C06936=1236.109,-121.710,-34.908,179.405,5.236,149.086
C06937=1236.114,-121.960,-34.900,179.403,5.236,149.087
C06938=1236.120,-122.210,-34.889,179.401,5.236,149.088
C06939=1236.125,-122.459,-34.879,179.399,5.236,149.088
C06940=1236.130,-122.709,-34.869,179.396,5.236,149.089
C06941=1236.136,-122.959,-34.860,179.394,5.236,149.090
C06942=1236.141,-123.209,-34.849,179.392,5.237,149.090
C06943=1236.145,-123.459,-34.840,179.389,5.236,149.091
C06944=1236.151,-123.708,-34.829,179.387,5.237,149.092
C06945=1236.156,-123.958,-34.820,179.384,5.236,149.093
C06946=1236.162,-124.208,-34.810,179.382,5.237,149.093
C06947=1236.167,-124.457,-34.800,179.380,5.236,149.094
C06948=1236.172,-124.707,-34.790,179.378,5.236,149.094
C06949=1236.178,-124.957,-34.781,179.375,5.236,149.095
C06950=1236.183,-125.207,-34.770,179.373,5.236,149.096
C06951=1236.188,-125.456,-34.761,179.371,5.236,149.097
C06952=1236.193,-125.706,-34.750,179.368,5.236,149.097
C06953=1236.198,-125.956,-34.741,179.366,5.236,149.098
C06954=1235.777,-125.967,-34.776,179.362,5.240,149.100
C06955=1235.771,-125.717,-34.786,179.364,5.239,149.099
C06956=1235.766,-125.467,-34.795,179.367,5.240,149.099
C06957=1235.760,-125.218,-34.806,179.369,5.240,149.098
C06958=1235.756,-124.968,-34.816,179.371,5.239,149.097
C06959=1235.750,-124.718,-34.825,179.373,5.240,149.097
C06960=1235.745,-124.468,-34.835,179.375,5.239,149.096
C06961=1235.740,-124.219,-34.845,179.378,5.240,149.095
C06962=1235.735,-123.969,-34.855,179.380,5.239,149.094
C06963=1235.730,-123.719,-34.864,179.383,5.240,149.094
C06964=1235.724,-123.469,-34.875,179.385,5.240,149.093
C06965=1235.719,-123.220,-34.885,179.387,5.239,149.093
C06966=1235.714,-122.970,-34.895,179.389,5.240,149.092
C06967=1235.708,-122.720,-34.904,179.391,5.239,149.091
C06968=1235.703,-122.470,-34.914,179.394,5.240,149.090
C06969=1235.698,-122.221,-34.924,179.396,5.239,149.090
C06970=1235.693,-121.971,-34.935,179.399,5.240,149.089
C06971=1235.688,-121.721,-34.944,179.401,5.240,149.088
C06972=1235.682,-121.471,-34.954,179.404,5.240,149.087
C06973=1235.677,-121.222,-34.964,179.406,5.240,149.087
C06974=1235.672,-120.972,-34.974,179.408,5.239,149.086
C06975=1235.667,-120.722,-34.984,179.410,5.240,149.086
C06976=1235.661,-120.473,-34.994,179.412,5.240,149.085
C06977=1235.656,-120.222,-35.004,179.415,5.240,149.084
C06978=1235.651,-119.973,-35.014,179.417,5.240,149.083
C06979=1235.645,-119.723,-35.024,179.420,5.240,149.083
C06980=1235.640,-119.474,-35.034,179.422,5.240,149.082
C06981=1235.635,-119.223,-35.044,179.424,5.240,149.081
C06982=1235.630,-118.974,-35.054,179.426,5.240,149.081
C06983=1235.624,-118.724,-35.065,179.429,5.239,149.080
C06984=1235.620,-118.474,-35.074,179.431,5.240,149.079
C06985=1235.614,-118.224,-35.084,179.433,5.240,149.078
C06986=1235.608,-117.975,-35.094,179.435,5.240,149.078
C06987=1235.604,-117.725,-35.104,179.438,5.240,149.077
C06988=1235.599,-117.475,-35.115,179.440,5.240,149.076
C06989=1235.593,-117.226,-35.125,179.442,5.240,149.076
C06990=1235.588,-116.975,-35.135,179.445,5.240,149.075
C06991=1235.583,-116.726,-35.145,179.447,5.240,149.074
C06992=1235.578,-116.477,-35.155,179.449,5.240,149.074
C06993=1235.573,-116.226,-35.166,179.452,5.240,149.073
C06994=1235.567,-115.977,-35.176,179.454,5.240,149.072
C06995=1235.562,-115.728,-35.186,179.457,5.240,149.071
C06996=1235.557,-115.477,-35.196,179.459,5.240,149.071
C06997=1235.552,-115.228,-35.206,179.461,5.240,149.070
C06998=1235.546,-114.978,-35.217,179.464,5.240,149.069
C06999=1235.542,-114.728,-35.226,179.466,5.240,149.069
C07000=1235.536,-114.479,-35.237,179.468,5.240,149.068
C07001=1235.530,-114.229,-35.247,179.471,5.241,149.067
C07002=1235.525,-113.979,-35.257,179.473,5.240,149.067
C07003=1235.520,-113.730,-35.268,179.475,5.240,149.066
C07004=1235.515,-113.479,-35.278,179.477,5.241,149.065
C07005=1235.510,-113.230,-35.288,179.479,5.240,149.065
C07006=1235.504,-112.981,-35.298,179.482,5.241,149.064
C07007=1235.499,-112.730,-35.309,179.484,5.240,149.063
C07008=1235.494,-112.481,-35.319,179.487,5.241,149.062
C07009=1235.488,-112.231,-35.329,179.489,5.240,149.062
C07010=1235.484,-111.981,-35.339,179.492,5.241,149.061
C07011=1235.478,-111.732,-35.349,179.494,5.240,149.060
C07012=1235.473,-111.481,-35.360,179.496,5.240,149.060
C07013=1235.468,-111.232,-35.370,179.499,5.240,149.059
C07014=1235.462,-110.982,-35.380,179.501,5.240,149.058
C07015=1235.457,-110.732,-35.391,179.503,5.241,149.057
C07016=1235.452,-110.483,-35.401,179.505,5.240,149.057
C07017=1235.447,-110.232,-35.412,179.508,5.241,149.056
C07018=1235.442,-109.983,-35.421,179.510,5.241,149.055
C07019=1235.437,-109.734,-35.433,179.512,5.241,149.055
C07020=1235.431,-109.484,-35.443,179.514,5.241,149.054
C07021=1235.426,-109.234,-35.453,179.517,5.241,149.053
C07022=1235.421,-108.984,-35.464,179.519,5.241,149.053
C07023=1235.415,-108.735,-35.474,179.521,5.240,149.052
C07024=1235.410,-108.484,-35.484,179.524,5.241,149.051
C07025=1235.405,-108.235,-35.494,179.526,5.240,149.050
C07026=1235.400,-107.985,-35.506,179.529,5.241,149.050
C07027=1235.395,-107.736,-35.515,179.531,5.241,149.049
C07028=1235.389,-107.486,-35.526,179.534,5.241,149.048
C07029=1235.384,-107.236,-35.536,179.536,5.241,149.048
C07030=1235.379,-106.987,-35.546,179.538,5.241,149.047
C07031=1235.374,-106.737,-35.558,179.540,5.241,149.046
C07032=1235.369,-106.487,-35.568,179.543,5.241,149.045
C07033=1235.364,-106.237,-35.578,179.545,5.241,149.045
C07034=1235.358,-105.988,-35.589,179.548,5.241,149.044
C07035=1235.353,-105.737,-35.599,179.550,5.241,149.043
C07036=1235.348,-105.489,-35.610,179.552,5.240,149.043
C07037=1235.343,-105.238,-35.621,179.555,5.241,149.042
C07038=1235.337,-104.989,-35.631,179.557,5.241,149.041
C07039=1235.332,-104.738,-35.642,179.559,5.241,149.041
C07040=1235.327,-104.490,-35.652,179.561,5.241,149.040
C07041=1235.322,-104.239,-35.663,179.564,5.241,149.039
C07042=1235.316,-103.990,-35.673,179.566,5.241,149.039
C07043=1235.311,-103.740,-35.684,179.569,5.242,149.038
C07044=1235.306,-103.491,-35.695,179.571,5.241,149.037
C07045=1235.301,-103.240,-35.705,179.573,5.242,149.036
C07046=1235.295,-102.991,-35.716,179.575,5.241,149.036
C07047=1235.291,-102.741,-35.727,179.578,5.242,149.035
C07048=1235.285,-102.492,-35.737,179.580,5.241,149.034
C07049=1235.280,-102.241,-35.748,179.582,5.241,149.034
C07050=1235.275,-101.992,-35.759,179.585,5.241,149.033
C07051=1235.270,-101.742,-35.769,179.587,5.241,149.032
C07052=1235.264,-101.493,-35.779,179.590,5.242,149.031
C07053=1235.259,-101.243,-35.791,179.592,5.241,149.031
C07054=1235.254,-100.994,-35.801,179.595,5.242,149.030
C07055=1235.248,-100.723,-35.813,179.597,5.241,149.029
C07056=1235.243,-100.451,-35.824,179.599,5.242,149.029
C07057=1235.237,-100.181,-35.836,179.602,5.242,149.028
C07058=1235.231,-99.909,-35.847,179.605,5.241,149.027
C07059=1235.226,-99.660,-35.859,179.607,5.242,149.026
C07060=1235.221,-99.410,-35.869,179.609,5.242,149.025
C07061=1235.216,-99.161,-35.880,179.612,5.242,149.025
C07062=1235.210,-98.911,-35.890,179.614,5.242,149.024
C07063=1235.205,-98.661,-35.901,179.616,5.241,149.023
C07064=1235.201,-98.411,-35.912,179.619,5.242,149.023
C07065=1235.195,-98.162,-35.922,179.621,5.241,149.022
C07066=1235.190,-97.912,-35.934,179.624,5.242,149.021
C07067=1235.185,-97.662,-35.944,179.626,5.241,149.020
C07068=1235.180,-97.413,-35.955,179.628,5.242,149.020
C07069=1235.174,-97.163,-35.966,179.630,5.242,149.019
C07070=1235.169,-96.913,-35.977,179.633,5.242,149.018
C07071=1235.164,-96.663,-35.988,179.635,5.242,149.018
C07072=1235.159,-96.414,-35.999,179.638,5.242,149.017
C07073=1235.154,-96.164,-36.009,179.640,5.242,149.016
C07074=1235.148,-95.915,-36.020,179.643,5.242,149.016
C07075=1235.143,-95.664,-36.032,179.645,5.242,149.015
C07076=1235.138,-95.415,-36.043,179.647,5.242,149.014
C07077=1235.132,-95.165,-36.053,179.650,5.242,149.013
C07078=1235.128,-94.916,-36.064,179.652,5.242,149.013
C07079=1235.122,-94.666,-36.075,179.654,5.242,149.012
C07080=1235.117,-94.417,-36.086,179.656,5.242,149.011
C07081=1235.112,-94.166,-36.097,179.659,5.242,149.011
C07082=1235.106,-93.917,-36.108,179.661,5.242,149.010
C07083=1235.101,-93.667,-36.118,179.664,5.242,149.009
C07084=1235.097,-93.417,-36.130,179.666,5.242,149.008
C07085=1235.091,-93.168,-36.140,179.669,5.242,149.008
C07086=1235.086,-92.918,-36.152,179.671,5.242,149.007
C07087=1235.081,-92.668,-36.163,179.673,5.242,149.006
C07088=1235.075,-92.418,-36.173,179.675,5.242,149.006
C07089=1235.071,-92.169,-36.185,179.678,5.243,149.005
C07090=1235.065,-91.918,-36.196,179.680,5.242,149.004
C07091=1235.060,-91.669,-36.207,179.683,5.243,149.003
C07092=1235.055,-91.420,-36.218,179.685,5.243,149.003
C07093=1235.049,-91.170,-36.228,179.687,5.243,149.002
C07094=1235.045,-90.921,-36.240,179.689,5.243,149.001
C07095=1235.039,-90.670,-36.251,179.692,5.243,149.001
C07096=1235.034,-90.420,-36.262,179.694,5.243,149.000
C07097=1235.029,-90.171,-36.273,179.697,5.243,148.999
C07098=1235.023,-89.921,-36.284,179.699,5.243,148.999
C07099=1235.019,-89.671,-36.295,179.702,5.243,148.998
C07100=1235.013,-89.422,-36.306,179.704,5.243,148.997
C07101=1235.008,-89.172,-36.317,179.707,5.243,148.996
C07102=1235.003,-88.922,-36.329,179.709,5.243,148.996
C07103=1234.998,-88.673,-36.340,179.711,5.242,148.995
C07104=1234.993,-88.423,-36.350,179.714,5.243,148.994
C07105=1234.987,-88.173,-36.362,179.716,5.243,148.993
C07106=1234.982,-87.924,-36.373,179.718,5.243,148.993
C07107=1234.977,-87.675,-36.384,179.720,5.243,148.992
C07108=1234.972,-87.424,-36.395,179.723,5.243,148.991
C07109=1234.967,-87.174,-36.407,179.725,5.243,148.991
C07110=1234.961,-86.925,-36.418,179.728,5.243,148.990
C07111=1234.957,-86.676,-36.429,179.730,5.243,148.989
C07112=1234.951,-86.425,-36.440,179.733,5.243,148.988
C07113=1234.946,-86.176,-36.452,179.735,5.243,148.988
C07114=1234.941,-85.927,-36.462,179.737,5.243,148.987
C07115=1234.936,-85.677,-36.474,179.740,5.243,148.986
C07116=1234.931,-85.427,-36.485,179.742,5.244,148.986
C07117=1234.925,-85.177,-36.497,179.744,5.243,148.985
C07118=1234.920,-84.928,-36.508,179.747,5.244,148.984
C07119=1234.915,-84.678,-36.519,179.749,5.243,148.983
C07120=1234.910,-84.428,-36.531,179.752,5.244,148.983
C07121=1234.905,-84.178,-36.541,179.754,5.243,148.982
C07122=1234.899,-83.929,-36.552,179.757,5.244,148.981
C07123=1234.894,-83.679,-36.564,179.759,5.244,148.981
C07124=1234.889,-83.429,-36.576,179.761,5.244,148.980
C07125=1234.884,-83.179,-36.587,179.763,5.244,148.979
C07126=1234.879,-82.931,-36.598,179.766,5.244,148.979
C07127=1234.874,-82.681,-36.610,179.768,5.244,148.978
C07128=1234.868,-82.430,-36.621,179.771,5.244,148.977
C07129=1234.864,-82.181,-36.632,179.773,5.244,148.976
C07130=1234.858,-81.931,-36.644,179.776,5.244,148.976
C07131=1234.853,-81.682,-36.655,179.778,5.244,148.975
C07132=1234.847,-81.432,-36.667,179.780,5.244,148.974
C07133=1234.843,-81.182,-36.678,179.782,5.244,148.974
C07134=1234.838,-80.933,-36.689,179.785,5.245,148.973
C07135=1234.833,-80.683,-36.701,179.787,5.244,148.972
C07136=1234.827,-80.434,-36.712,179.790,5.245,148.971
C07137=1234.822,-80.183,-36.723,179.792,5.244,148.971
C07138=1234.817,-79.934,-36.735,179.795,5.245,148.970
C07139=1234.811,-79.684,-36.747,179.797,5.245,148.969
C07140=1234.807,-79.434,-36.758,179.799,5.245,148.969
C07141=1234.801,-79.184,-36.770,179.801,5.245,148.968
C07142=1234.796,-78.935,-36.781,179.804,5.245,148.967
C07143=1234.791,-78.685,-36.793,179.806,5.245,148.966
C07144=1234.786,-78.436,-36.804,179.809,5.245,148.966
C07145=1234.780,-78.186,-36.816,179.811,5.245,148.965
C07146=1234.776,-77.936,-36.827,179.814,5.245,148.964
C07147=1234.770,-77.686,-36.839,179.816,5.245,148.964
C07148=1234.765,-77.437,-36.850,179.818,5.245,148.963
C07149=1234.760,-77.187,-36.862,179.821,5.245,148.962
C07150=1234.755,-76.938,-36.873,179.823,5.246,148.961
C07151=1234.749,-76.688,-36.885,179.825,5.245,148.961
C07152=1234.745,-76.438,-36.896,179.828,5.246,148.960
C07153=1234.739,-76.188,-36.908,179.830,5.245,148.959
C07154=1234.734,-75.938,-36.920,179.833,5.246,148.959
C07155=1234.729,-75.689,-36.931,179.835,5.245,148.958
C07156=1234.723,-75.439,-36.943,179.837,5.246,148.957
C07157=1234.718,-75.190,-36.954,179.840,5.246,148.957
C07158=1234.713,-74.940,-36.967,179.843,5.246,148.956
C07159=1234.708,-74.669,-36.979,179.845,5.245,148.955
C07160=1234.702,-74.400,-36.991,179.848,5.246,148.954
C07161=1234.697,-74.129,-37.004,179.850,5.246,148.953
C07162=1234.691,-73.858,-37.017,179.853,5.246,148.953
C07163=1234.686,-73.610,-37.028,179.855,5.246,148.952
C07164=1234.681,-73.360,-37.040,179.858,5.246,148.951
C07165=1234.675,-73.110,-37.052,179.860,5.246,148.950
C07166=1234.670,-72.861,-37.063,179.862,5.246,148.950
C07167=1234.665,-72.611,-37.075,179.865,5.246,148.949
C07168=1234.660,-72.361,-37.087,179.867,5.246,148.948
C07169=1234.655,-72.111,-37.098,179.870,5.246,148.948
C07170=1234.650,-71.862,-37.111,179.872,5.246,148.947
C07171=1234.645,-71.612,-37.122,179.874,5.247,148.946
C07172=1234.640,-71.362,-37.134,179.877,5.246,148.945
C07173=1234.634,-71.112,-37.146,179.879,5.247,148.945
C07174=1234.629,-70.863,-37.157,179.881,5.246,148.944
C07175=1234.623,-70.613,-37.169,179.884,5.247,148.943
C07176=1234.618,-70.364,-37.182,179.886,5.247,148.943
C07177=1234.614,-70.115,-37.193,179.889,5.247,148.942
C07178=1234.608,-69.865,-37.205,179.891,5.247,148.941
C07179=1234.603,-69.615,-37.217,179.894,5.247,148.940
C07180=1234.598,-69.365,-37.228,179.896,5.247,148.940
C07181=1234.593,-69.116,-37.240,179.898,5.247,148.939
C07182=1234.588,-68.866,-37.252,179.900,5.247,148.938
C07183=1234.583,-68.616,-37.264,179.903,5.247,148.938
C07184=1234.577,-68.366,-37.276,179.905,5.247,148.937
C07185=1234.572,-68.117,-37.288,179.908,5.248,148.936
C07186=1234.567,-67.867,-37.300,179.911,5.248,148.935
C07187=1234.562,-67.617,-37.311,179.913,5.247,148.935
C07188=1234.557,-67.368,-37.324,179.916,5.248,148.934
C07189=1234.552,-67.118,-37.336,179.918,5.247,148.933
C07190=1234.547,-66.868,-37.347,179.920,5.248,148.932
C07191=1234.541,-66.619,-37.359,179.923,5.248,148.932
C07192=1234.536,-66.369,-37.372,179.925,5.248,148.931
C07193=1234.531,-66.119,-37.383,179.927,5.248,148.930
C07194=1234.526,-65.870,-37.395,179.930,5.248,148.930
C07195=1234.521,-65.620,-37.407,179.932,5.248,148.929
C07196=1234.516,-65.370,-37.419,179.935,5.248,148.928
C07197=1234.510,-65.120,-37.431,179.937,5.248,148.928
C07198=1234.505,-64.871,-37.444,179.940,5.248,148.927
C07199=1234.500,-64.622,-37.455,179.942,5.248,148.926
C07200=1234.495,-64.372,-37.468,179.944,5.249,148.925
C07201=1234.490,-64.122,-37.479,179.946,5.248,148.925
C07202=1234.484,-63.872,-37.491,179.949,5.249,148.924
C07203=1234.480,-63.623,-37.503,179.951,5.248,148.923
C07204=1234.475,-63.373,-37.515,179.954,5.249,148.923
C07205=1234.469,-63.123,-37.527,179.956,5.249,148.922
C07206=1234.464,-62.874,-37.540,179.959,5.249,148.921
C07207=1234.459,-62.624,-37.552,179.961,5.250,148.920
C07208=1234.454,-62.375,-37.564,179.963,5.249,148.920
C07209=1234.449,-62.125,-37.576,179.966,5.249,148.919
C07210=1234.444,-61.876,-37.588,179.969,5.249,148.918
C07211=1234.439,-61.625,-37.600,179.971,5.249,148.917
C07212=1234.434,-61.376,-37.613,179.973,5.249,148.917
C07213=1234.428,-61.126,-37.625,179.976,5.250,148.916
C07214=1234.423,-60.876,-37.637,179.978,5.249,148.915
C07215=1234.419,-60.627,-37.649,179.981,5.250,148.915
C07216=1234.413,-60.377,-37.661,179.983,5.249,148.914
C07217=1234.408,-60.128,-37.673,179.985,5.250,148.913
C07218=1234.403,-59.878,-37.685,179.988,5.250,148.912
C07219=1234.397,-59.629,-37.698,179.990,5.250,148.912
C07220=1234.392,-59.379,-37.710,179.993,5.251,148.911
C07221=1234.387,-59.129,-37.722,179.995,5.250,148.910
C07222=1234.382,-58.880,-37.735,179.998,5.251,148.910
C07223=1234.378,-58.630,-37.746,180.000,5.250,148.909
C07224=1234.373,-58.380,-37.759,-179.998,5.251,148.908
C07225=1234.367,-58.130,-37.771,-179.995,5.251,148.908
C07226=1234.362,-57.881,-37.784,-179.993,5.251,148.907
C07227=1234.357,-57.631,-37.795,-179.991,5.251,148.906
C07228=1234.351,-57.382,-37.808,-179.988,5.251,148.905
C07229=1234.346,-57.132,-37.820,-179.985,5.250,148.904
C07230=1234.341,-56.883,-37.833,-179.983,5.251,148.904
C07231=1234.336,-56.633,-37.845,-179.981,5.251,148.903
C07232=1234.331,-56.383,-37.857,-179.978,5.251,148.902
C07233=1234.326,-56.133,-37.870,-179.975,5.252,148.902
C07234=1234.320,-55.883,-37.882,-179.973,5.251,148.901
C07235=1234.315,-55.634,-37.894,-179.971,5.252,148.900
C07236=1234.310,-55.385,-37.907,-179.969,5.251,148.900
C07237=1234.305,-55.135,-37.918,-179.966,5.252,148.899
C07238=1234.301,-54.885,-37.931,-179.964,5.252,148.898
C07239=1234.296,-54.636,-37.944,-179.961,5.252,148.897
C07240=1234.290,-54.386,-37.956,-179.959,5.252,148.897
C07241=1234.285,-54.137,-37.968,-179.956,5.252,148.896
C07242=1234.280,-53.887,-37.981,-179.954,5.252,148.895
C07243=1234.275,-53.637,-37.993,-179.952,5.252,148.895
C07244=1234.270,-53.387,-38.006,-179.949,5.253,148.894
C07245=1234.265,-53.138,-38.018,-179.947,5.253,148.893
C07246=1234.260,-52.888,-38.030,-179.944,5.253,148.893
C07247=1234.254,-52.639,-38.043,-179.942,5.253,148.892
C07248=1234.249,-52.389,-38.056,-179.939,5.253,148.891
C07249=1234.245,-52.139,-38.068,-179.937,5.252,148.890
C07250=1234.239,-51.889,-38.080,-179.934,5.253,148.889
C07251=1234.234,-51.640,-38.093,-179.932,5.253,148.889
C07252=1234.228,-51.390,-38.106,-179.929,5.253,148.888
C07253=1234.223,-51.141,-38.118,-179.927,5.254,148.887
C07254=1234.218,-50.891,-38.131,-179.925,5.253,148.887
C07255=1234.213,-50.641,-38.144,-179.922,5.254,148.886
C07256=1234.208,-50.392,-38.156,-179.920,5.253,148.885
C07257=1234.203,-50.143,-38.169,-179.917,5.254,148.885
C07258=1234.198,-49.893,-38.181,-179.915,5.254,148.884
C07259=1234.193,-49.643,-38.194,-179.913,5.254,148.883
C07260=1234.188,-49.393,-38.206,-179.910,5.254,148.882
C07261=1234.183,-49.144,-38.219,-179.908,5.254,148.882
C07262=1234.178,-48.895,-38.232,-179.905,5.255,148.881
C07263=1234.172,-48.624,-38.245,-179.903,5.254,148.880
C07264=1234.167,-48.354,-38.259,-179.900,5.255,148.879
C07265=1234.161,-48.085,-38.272,-179.897,5.255,148.879
C07266=1234.155,-47.815,-38.286,-179.895,5.254,148.878
C07267=1234.150,-47.566,-38.299,-179.892,5.255,148.877
C07268=1234.146,-47.316,-38.312,-179.890,5.255,148.876
C07269=1234.140,-47.066,-38.324,-179.887,5.255,148.876
C07270=1234.135,-46.817,-38.336,-179.885,5.256,148.875
C07271=1234.130,-46.567,-38.349,-179.882,5.255,148.874
C07272=1234.125,-46.317,-38.363,-179.880,5.256,148.874
C07273=1234.120,-46.068,-38.375,-179.878,5.255,148.873
C07274=1234.115,-45.818,-38.388,-179.875,5.256,148.872
C07275=1234.109,-45.569,-38.400,-179.873,5.256,148.871
C07276=1234.105,-45.319,-38.413,-179.870,5.256,148.871
C07277=1234.100,-45.070,-38.426,-179.868,5.257,148.870
C07278=1234.094,-44.820,-38.439,-179.866,5.256,148.869
C07279=1234.089,-44.569,-38.451,-179.863,5.257,148.869
C07280=1234.084,-44.320,-38.464,-179.861,5.256,148.868
C07281=1234.079,-44.071,-38.477,-179.858,5.257,148.867
C07282=1234.074,-43.821,-38.489,-179.856,5.257,148.867
C07283=1234.068,-43.571,-38.503,-179.853,5.257,148.866
C07284=1234.063,-43.322,-38.515,-179.850,5.257,148.865
C07285=1234.058,-43.072,-38.528,-179.848,5.257,148.864
C07286=1234.054,-42.822,-38.541,-179.845,5.257,148.863
C07287=1234.048,-42.573,-38.554,-179.843,5.257,148.863
C07288=1234.043,-42.324,-38.567,-179.841,5.258,148.862
C07289=1234.038,-42.074,-38.580,-179.839,5.257,148.861
C07290=1234.033,-41.824,-38.592,-179.836,5.258,148.861
C07291=1234.027,-41.575,-38.605,-179.833,5.258,148.860
C07292=1234.023,-41.325,-38.618,-179.831,5.258,148.859
C07293=1234.018,-41.075,-38.631,-179.829,5.258,148.859
C07294=1234.012,-40.826,-38.644,-179.826,5.258,148.858
C07295=1234.007,-40.576,-38.657,-179.824,5.259,148.857
C07296=1234.002,-40.327,-38.671,-179.821,5.259,148.856
C07297=1233.997,-40.078,-38.683,-179.819,5.259,148.856
C07298=1233.993,-39.828,-38.696,-179.816,5.259,148.855
C07299=1233.987,-39.578,-38.709,-179.814,5.259,148.854
C07300=1233.982,-39.328,-38.722,-179.811,5.259,148.853
